			(* Löschen der Kraftwerte in den beiden IST-Einpresskurven *)
			FOR i16_ku_nr := 0  TO i_MAX_KURVEN BY 1DO
				FOR i16_mp_nr := 0  TO i_MAX_MESSPUNKTE BY 1DO
					st_ausgabe.st_kurve[i16_ku_nr].arr_kraft_ist[i16_mp_nr] := 0;
					st_ausgabe.st_kurve[i16_ku_nr].arr_weg_ist[i16_mp_nr] := 0;
				END_FOR
			END_FOR

			(* Löschen der Kraftwerte in allen Stützkurven*)
			IF st_einpressen.st_einstellungen.enu_modus = STUETZKURVE THEN
				FOR i16_ku_nr := 0  TO i_MAX_KURVEN BY 1DO
					FOR i16_mp_nr := 0  TO i_MAX_MESSPUNKTE BY 1DO
						st_ausgabe.st_kurve[i16_ku_nr].arr_kraft_stuetz[i16_mp_nr] := 0;
						st_ausgabe.st_kurve[i16_ku_nr].arr_weg_stuetz[i16_mp_nr] := 0;
					END_FOR
				END_FOR
			END_IF
		END_IF

		(* Hochzählen mit der Anzahl der bestückten Pins *)
		i16_pin_nr := ST_Virtuelle_Masterachse.i16_bestueckposzaehler;
		(* Abfrage Array-Grösse auf Überlauf *)
		IF i16_pin_nr > i_MAX_KURVEN THEN
			i16_pin_nr := 0;
		END_IF

		(* Die Messpunkte werden gradgenau aufgenommen und entsprechen deshalb den Winkelgraden der Bestückachse *)
		i16_mp_nr := ui_akt_pos_bestueckachse;

		CASE st_einpressen.st_einstellungen.enu_modus OF
			KEIN_MODUS:	(* Fehler Auswahl Einpressmodus *)
				sm_fehler_einpressmodus := TRUE;
				fb_state_entry.i16_next_step := FEHLER;

			FMAX:	(* Einpressen mit Überwachung auf Maximalkraft und Sicherheitsabfrage der Minimalkraft*)
				(*st_einpressen.st_einstellungen.lr_minkraft_einpressen := 12.0;*)
				IF  lr_kraft_n > st_ausgabe.st_ergebnisse.lr_maxkraft_einpressen THEN
					st_ausgabe.st_ergebnisse.lr_maxkraft_einpressen := lr_kraft_n;
				END_IF
				(* Fehlerfall: Voreingestellte Maximalkraft überschritten nur im Automatik Betrieb *)
				IF  gi16_betriebsart = AUTO AND lr_kraft_n > lr_help_maxkraft_einpressen THEN		(*st_einpressen.st_einstellungen.lr_maxkraft_einpressen*)
					sm_aktkraft_groesser_maxkraft_einpressen := TRUE;
					fb_state_entry.i16_next_step := FEHLER;
				END_IF

				(* Fehlerfall: Voreingestellte Minimalkraft unterschritten *)
				IF	lr_weg_grad =0 THEN
					st_ausgabe.st_ergebnisse.lr_maxkraft_einpres_proHub:=0;
				END_IF
				IF  lr_kraft_n > st_ausgabe.st_ergebnisse.lr_maxkraft_einpres_proHub THEN
					st_ausgabe.st_ergebnisse.lr_maxkraft_einpres_proHub:=lr_kraft_n;
				END_IF

				IF	gi16_betriebsart = AUTO AND
					st_einpressen.st_einstellungen.lr_minkraft_einpressen > 0 AND
					nockenschaltwerk_bestueckachse.fb.arr_spur[SP_BESTUECKSCHIEBERHUB ] AND
					st_ausgabe.st_ergebnisse.lr_maxkraft_einpres_proHub < st_einpressen.st_einstellungen.lr_minkraft_einpressen	THEN
					i16_merker:=i16_merker+1;
					(*	sm_aktkraft_kleiner_minkraft_einpressen := TRUE;
						fb_state_entry.i16_next_step := FEHLER;*)
				END_IF

				(* Aufzeichnen der Überlaufkraft nach einem Einpressfehler *)
				IF  lr_kraft_n > st_ausgabe.st_ergebnisse.lr_ueberlaufkraft THEN
					st_ausgabe.st_ergebnisse.lr_ueberlaufkraft := lr_kraft_n;
				END_IF

			FMIN_FMAX:	(* Einpressen mit Überwachung von Minimal- und Maximalkraft. Der Weg spielt hier keine Rolle! *)
				(* Aktuelle Kraft gradgenau einlesen *)
				IF st_ausgabe.st_kurve[i16_pin_nr].arr_kraft_ist[i16_mp_nr] = 0 THEN
					(* Einmalig den aktuellen Kraftwert eintragen, wenn Messpunkt im Array noch leer ist *)
					st_ausgabe.st_kurve[i16_pin_nr].arr_kraft_ist[i16_mp_nr] := lr_kraft_n;
				END_IF

				(* Aufnehmen der maximal aufgetretenen Kraft *)
				IF st_ausgabe.st_kurve[i16_pin_nr].arr_kraft_ist[i16_mp_nr] > st_ausgabe.st_ergebnisse.lr_maxkraft_einpressen THEN
					st_ausgabe.st_ergebnisse.lr_maxkraft_einpressen := st_ausgabe.st_kurve[i16_pin_nr].arr_kraft_ist[i16_mp_nr];
				END_IF

				(* Fehlerfall: Überwachen der Maximalkraft beim Aufnahmehub *)
				IF 	nockenschaltwerk_bestueckachse.fb.arr_spur[SP_AUFNAHMEHUB ] AND
					st_ausgabe.st_kurve[i16_pin_nr].arr_kraft_ist[i16_mp_nr] > 0
					THEN
						IF st_ausgabe.st_kurve[i16_pin_nr].arr_kraft_ist[i16_mp_nr] > st_einpressen.st_einstellungen.lr_maxkraft_aufnahme THEN
							st_einpressen.st_einstellungen.lr_maxkraft_aufnahme := st_ausgabe.st_kurve[i16_pin_nr].arr_kraft_ist[i16_mp_nr];
							sm_aktkraft_groesser_maxkraft_aufnahme := TRUE;
							fb_state_entry.i16_next_step := FEHLER;
						END_IF
				END_IF

				(* Fehlerfall: Überwachen der Maximalkraft beim Auftreffen des Pins auf den Isolierkörper *)
				IF 	nockenschaltwerk_bestueckachse.fb.arr_spur[SP_EINPRESSHUB ] AND
					st_ausgabe.st_kurve[i16_pin_nr].arr_kraft_ist[i16_mp_nr] > 0
					THEN
						IF st_ausgabe.st_kurve[i16_pin_nr].arr_kraft_ist[i16_mp_nr] > st_einpressen.st_einstellungen.lr_maxkraft_einpressen THEN
							st_einpressen.st_einstellungen.lr_maxkraft_einpressen := st_ausgabe.st_kurve[i16_pin_nr].arr_kraft_ist[i16_mp_nr];
							sm_aktkraft_groesser_maxkraft_einpressen := TRUE;
							fb_state_entry.i16_next_step := FEHLER;
						END_IF
				END_IF

				(* Fehlerfall: Überwachen der Minimalkraft beim Einpresshub *)
				IF 	nockenschaltwerk_bestueckachse.fb.arr_spur[SP_MIN_KRAFT_EINPRESSEN ] AND
					st_ausgabe.st_kurve[i16_pin_nr].arr_kraft_ist[i16_mp_nr] > 0
					THEN
						IF st_ausgabe.st_kurve[i16_pin_nr].arr_kraft_ist[i16_mp_nr] < st_einpressen.st_einstellungen.lr_minkraft_einpressen THEN
							st_einpressen.st_einstellungen.lr_minkraft_einpressen := st_ausgabe.st_kurve[i16_pin_nr].arr_kraft_ist[i16_mp_nr];
							sm_aktkraft_kleiner_minkraft_einpressen := TRUE;
							fb_state_entry.i16_next_step := FEHLER;
						END_IF
				END_IF

			HUELLKURVE:	(* Einpressen mit Hüllkurve um Stützkurve*)
				(* Aktuelle Kraft in die Ist-Kurve einlesen *)
				IF st_ausgabe.st_kurve[i16_pin_nr].arr_kraft_ist[i16_mp_nr] = 0 THEN
					(* Einmalig den aktuellen Kraftwert eintragen, wenn Messpunkt im Array noch leer ist *)
					st_ausgabe.st_kurve[i16_pin_nr].arr_kraft_ist[i16_mp_nr] := lr_kraft_n;
				END_IF
				(* Aktuellen Weg in die Ist-Kurve einlesen, wobei in diesem Fall das Arrayelement dem aktuellen Winkel entspricht. *)
				IF st_ausgabe.st_kurve[i16_pin_nr].arr_weg_ist[i16_mp_nr] = 0 THEN
					(* Einmalig den aktuellen Wegwert eintragen, wenn Messpunkt im Array noch leer ist *)
					st_ausgabe.st_kurve[i16_pin_nr].arr_weg_ist[i16_mp_nr] := lr_weg_grad;
				END_IF

				(* Toleranzabfrage und Fehlerauswertung *)
				IF st_ausgabe.st_kurve[i16_pin_nr].arr_kraft_ist[i16_mp_nr] > 0 AND st_ausgabe.st_kurve[i16_pin_nr].arr_weg_ist[i16_mp_nr] > 0 THEN
					b_kraft_weg_in_mp_ok := FALSE;
					(* Werte sind gültig -> Abfrage , ob Kraft und Weg im Toleranzrechteck liegen. *)
					FOR i16_mp_nr := 0  TO i_MAX_MESSPUNKTE BY 1DO
						IF	st_ausgabe.st_kurve[i16_pin_nr].arr_kraft_ist[i16_mp_nr] >= (st_ausgabe.st_kurve[i16_pin_nr].arr_kraft_ist[i16_mp_nr] - st_einpressen.st_einstellungen.lr_delta_kraft) AND
							st_ausgabe.st_kurve[i16_pin_nr].arr_kraft_ist[i16_mp_nr] <= (st_ausgabe.st_kurve[i16_pin_nr].arr_kraft_ist[i16_mp_nr] + st_einpressen.st_einstellungen.lr_delta_kraft) AND
							st_ausgabe.st_kurve[i16_pin_nr].arr_weg_ist[i16_mp_nr] >= (st_ausgabe.st_kurve[i16_pin_nr].arr_weg_ist[i16_mp_nr] - st_einpressen.st_einstellungen.lr_delta_weg) AND
							st_ausgabe.st_kurve[i16_pin_nr].arr_weg_ist[i16_mp_nr] <= (st_ausgabe.st_kurve[i16_pin_nr].arr_weg_ist[i16_mp_nr] + st_einpressen.st_einstellungen.lr_delta_weg)
							THEN
								b_kraft_weg_in_mp_ok := TRUE;
								EXIT;
						ELSE
							b_kraft_weg_in_mp_ok := FALSE;
						END_IF
					END_FOR

					(* Fehlerfall: Aktueller Messpunkt liegt mit seiner Kraft oder seinem Weg nicht im Toleranzrechteck *)
					IF NOT b_kraft_weg_in_mp_ok THEN
						sm_kraft_weg_ausserhalb_huellkurve := TRUE;
						fb_state_entry.i16_next_step := FEHLER;
					END_IF
				END_IF

			STUETZKURVE:	(* Einlernen der Stützkurve *)
				(* Aktuelle Kraft in die Stuetzkurve einlesen *)
				IF st_ausgabe.st_kurve[i16_pin_nr].arr_kraft_stuetz[i16_mp_nr] = 0 THEN
					(* Einmalig den aktuellen Kraftwert eintragen, wenn Messpunkt im Array noch leer ist *)
					st_ausgabe.st_kurve[i16_pin_nr].arr_kraft_stuetz[i16_mp_nr] := lr_kraft_n;
				END_IF
				(* Aktuellen Weg in die Stuetzkurve einlesen, wobei in diesem Fall das Arrayelement dem aktuellen Winkel entspricht. *)
				IF st_ausgabe.st_kurve[i16_pin_nr].arr_weg_stuetz[i16_mp_nr] = 0 THEN
					(* Einmalig den aktuellen Wegwert eintragen, wenn Messpunkt im Array noch leer ist *)
					st_ausgabe.st_kurve[i16_pin_nr].arr_weg_stuetz[i16_mp_nr] := lr_weg_grad;
				END_IF
		END_CASE

		(* Manuelle Messbereichsumschaltung anhand des Einstellwertes für Maximalkraft beim Einpressen. *)
		IF gst_datensatz.st_band.st_einpressen.st_einstellungen.lr_maxkraft_einpressen > (i_KRAFTFAKTOR_MB1 * 0.75) THEN
			a_messbereich_1_oder_2 := TRUE;
		ELSE
			(* Automatische Messbereichsumschaltung, wenn die maximale Einpresskraft 75% des Messbereichsendwertes überschreitet. *)
			IF st_ausgabe.st_ergebnisse.lr_maxkraft_einpressen > (i_KRAFTFAKTOR_MB1 * 0.75) THEN
				a_messbereich_1_oder_2 := TRUE;
			END_IF
		END_IF

		(*-----------------------Weiterschaltbedingungen----------------------------*)
		IF NOT st_ctrl_in.b_start THEN
			(* Messbereichsanpassung nur, wenn die Krafteinstellung für maximale Einpresskraft es erlaubt. *)
			IF gst_datensatz.st_band.st_einpressen.st_einstellungen.lr_maxkraft_einpressen < (i_KRAFTFAKTOR_MB1 * 0.75) THEN
				(* Automatische Messbereichsumschaltung, wenn die maximale Einpresskraft 50% des Messbereichsendwertes unterschreitet. *)
				IF st_ausgabe.st_ergebnisse.lr_maxkraft_einpressen < (i_KRAFTFAKTOR_MB1 * 0.5) THEN
					a_messbereich_1_oder_2 := FALSE;
				END_IF
			END_IF
			a_start_messung := FALSE;
			fb_state_entry.i16_next_step := BEREIT;
		END_IF

(*=======================================================*)
	FEHLER:
		IF fb_state_entry.E THEN
			st_ctrl_out.b_fehler := TRUE;
			fb_ton_quitt.IN := FALSE;
		END_IF

		(* Aufzeichnen der Überlaufkraft nach einem Einpressfehler *)
		IF  lr_kraft_n > st_ausgabe.st_ergebnisse.lr_ueberlaufkraft THEN
			st_ausgabe.st_ergebnisse.lr_ueberlaufkraft := lr_kraft_n;
		END_IF

		(*-----------------------Weiterschaltbedingungen----------------------------*)
		IF st_ctrl_in.b_quitt AND NOT fb_state_entry.E THEN
			st_ctrl_out.b_fehler := FALSE;
			fb_ton_quitt.IN := TRUE;
		END_IF

		IF fb_ton_quitt.Q THEN
			fb_ton_quitt.IN := FALSE;
			fb_state_entry.i16_next_step := INIT;
		END_IF

(*=======================================================*)
	STOP:
		IF fb_state_entry.E THEN
			fb_ton_quitt.IN := FALSE;
		END_IF

		(*-----------------------Weiterschaltbedingungen----------------------------*)
		IF st_ctrl_in.b_quitt AND NOT fb_state_entry.E THEN
			fb_ton_quitt.IN := TRUE;
		END_IF

		IF fb_ton_quitt.Q THEN
			fb_ton_quitt.IN := FALSE;
			fb_state_entry.i16_next_step := INIT;
		END_IF
END_CASE

fb_state_entry(
	i16_next_step:= ,
	i16_pos:= 2,
	s_debugtext:= ,
	E=> , 
	X=> ,
	i16_step=> ,
	i16_last_step=> );

(* Fehlermeldungen und Betriebsmeldungen ab dem Startindex in die globalen Meldungsarrays schreiben *)
garr_stoermeldungen[st_config.i16_meld_startindex + 0] := sm_fehler_einpressmodus;
garr_stoermeldungen[st_config.i16_meld_startindex + 1] := sm_aktkraft_groesser_maxkraft_aufnahme;
garr_stoermeldungen[st_config.i16_meld_startindex + 2] := sm_aktkraft_groesser_maxkraft_einpressen;
garr_stoermeldungen[st_config.i16_meld_startindex + 3] := sm_aktkraft_kleiner_minkraft_einpressen;
garr_stoermeldungen[st_config.i16_meld_startindex + 4] := sm_kraft_weg_ausserhalb_huellkurve;
garr_stoermeldungen[st_config.i16_meld_startindex + 5] := sm_fehler_analogwert_kraftmessdose;
garr_stoermeldungen[st_config.i16_meld_startindex + 6] := sm_max_mb_ueberschritten;
garr_stoermeldungen[st_config.i16_meld_startindex + 7] := sm_max_einstell_mb_ueberschritten;
garr_stoermeldungen[st_config.i16_meld_startindex + 8] := FALSE;
garr_stoermeldungen[st_config.i16_meld_startindex + 9] := FALSE;
garr_stoermeldungen[st_config.i16_meld_startindex + 10] := FALSE;
garr_stoermeldungen[st_config.i16_meld_startindex + 11] := FALSE;
garr_stoermeldungen[st_config.i16_meld_startindex + 12] := FALSE;
garr_stoermeldungen[st_config.i16_meld_startindex + 13] := FALSE;
garr_stoermeldungen[st_config.i16_meld_startindex + 14] := FALSE;
garr_stoermeldungen[st_config.i16_meld_startindex + 15] := FALSE;
garr_stoermeldungen[st_config.i16_meld_startindex + 16] := FALSE;
garr_stoermeldungen[st_config.i16_meld_startindex + 17] := FALSE;
garr_stoermeldungen[st_config.i16_meld_startindex + 18] := FALSE;
garr_stoermeldungen[st_config.i16_meld_startindex + 19] := FALSE;

garr_betriebsmeldungen[st_config.i16_meld_startindex + 0] := FALSE;
garr_betriebsmeldungen[st_config.i16_meld_startindex + 1] := FALSE;
garr_betriebsmeldungen[st_config.i16_meld_startindex + 2] := FALSE;
garr_betriebsmeldungen[st_config.i16_meld_startindex + 3] := FALSE;
garr_betriebsmeldungen[st_config.i16_meld_startindex + 4] := FALSE;
garr_betriebsmeldungen[st_config.i16_meld_startindex + 5] := FALSE;
garr_betriebsmeldungen[st_config.i16_meld_startindex + 6] := FALSE;
garr_betriebsmeldungen[st_config.i16_meld_startindex + 7] := FALSE;
garr_betriebsmeldungen[st_config.i16_meld_startindex + 8] := FALSE;
garr_betriebsmeldungen[st_config.i16_meld_startindex + 9] := FALSE;
garr_betriebsmeldungen[st_config.i16_meld_startindex + 10] := FALSE;
garr_betriebsmeldungen[st_config.i16_meld_startindex + 11] := FALSE;
garr_betriebsmeldungen[st_config.i16_meld_startindex + 12] := FALSE;
garr_betriebsmeldungen[st_config.i16_meld_startindex + 13] := FALSE;
garr_betriebsmeldungen[st_config.i16_meld_startindex + 14] := FALSE;
garr_betriebsmeldungen[st_config.i16_meld_startindex + 15] := FALSE;
garr_betriebsmeldungen[st_config.i16_meld_startindex + 16] := FALSE;
garr_betriebsmeldungen[st_config.i16_meld_startindex + 17] := FALSE;
garr_betriebsmeldungen[st_config.i16_meld_startindex + 18] := FALSE;
garr_betriebsmeldungen[st_config.i16_meld_startindex + 19] := FALSE;
END_PROGRAM

(* POU EPT Lib/CamEditor/Verfahrberechnungen/ST_MFCalcConstPhase, ST *)
FUNCTION_BLOCK ST_MFCalcConstPhase
VAR_INPUT
	st_config								: struct_config;
	st_ctrl_in								: struct_ctrl_in;

	(* Kurvenscheibendaten *)
	udiTableId							: MC_CAM_ID;			(* Table-ID *)
	eMotionFunctionType					: MC_MotionFunctionType;	(*Bewegungsgesetz: MOTIONFUNCTYPE_POLYNOM5 etc.*)
	i16_startpunkt_edit_mf_tab				: INT;
	arr_db_mf_tab						: ARRAY[1..i_MAX_NUM_MFP] OF struct_db_motionfunctionpoint;	(* Vorgabe aus der Datenbank *)

	(* Bewegungsdaten an der Last *)
	lrVeloMax							: LREAL;	(*maximale Geschwindigkeit [mm/s] an der Last *)
	lrAccMax								: LREAL;	(*maximale Beschleunigung [mm/s²] an der Last *)
	lrDecMax							: LREAL;	(*maximale Beschleunigung [mm/s²] an der Last *)

	lrModuloValue 						: LREAL ;
END_VAR
VAR_IN_OUT
	st_AxisRefMaster						: AXIS_REF;
	st_AxisRefSlave						: AXIS_REF;
END_VAR
VAR_OUTPUT
	lrMasterVeloMax						: LREAL;	(* Maximum Master Velocity [°/s] *)
	lrMasterRotPerMinMax					: LREAL;	(* Maximum Master Rotations per Minute [1/min] *)
	st_ctrl_out							: struct_ctrl_out;
END_VAR
VAR
	st_sm						 		: struct_cameditor_meldungen;
	fb_state_entry							: ST_StateEntry;
	fb_ton_quitt							: TON;
	fb_ton_wz							: TON;

	stMotionFunctionPointDummy			: MC_MotionFunctionPoint;	(* Dummy-Punkt *)
(*	TYPE MC_MotionFunctionPoint :
		STRUCT
		    PointIndex        		: MC_MotionFunctionPoint_ID;
		    FunctionType   		: MC_MotionFunctionType;
		    PointType         		: MC_MotionPointType;
		    RelIndexNextPoint 	: MC_MotionFunctionPoint_ID;
		    MasterPos         		: LREAL; (* X *)
		    SlavePos          		: LREAL; (* Y *)
		    SlaveVelo         		: LREAL; (* Y' *)
		    SlaveAcc          		: LREAL; (* Y'' *)
		    SlaveJerk         		: LREAL; (* Y''' *)
		END_STRUCT
	END_TYPE
*)

	(*Motion Function runterschreiben an NC*)
	astWriteMotionFunction 				: ARRAY[1..i_MAX_NUM_MFP] OF MC_MotionFunctionPoint;
	stWriteMFCamTableRef				: MC_CAM_Ref;	(*Definition Zieltabelle*)
	fbCamTableSelect					: MC_CamTableSelect;
	fbWriteMF							: MC_WriteMotionFunction;
	b_cam_table_select_periodic			: BOOL := FALSE;
	b_cam_table_select_master_absolute	: BOOL := FALSE;
	b_cam_table_select_slave_absolute		: BOOL := FALSE;

	(*Motion Function hochladen von NC*)
	fbReadMF							: MC_ReadMotionFunction;
	stReadMFCamTableRef				: MC_CAM_Ref;	(*Definition Zieltabelle*)
	astReadMotionFunction 				: ARRAY[0..i_MAX_NUM_MFP] OF MC_MotionFunctionPoint;

	(*Berechnung Konstantfahrphase*)
	fbMFcalcConstVelo					: ST_MFcalcConstVelo;	(*Baustein zur Berechnung, ob eine Konstantfahphase möglich ist*)
	stDataCalcConstVelo 					: ARRAY[1..4] OF MC_MotionFunctionPoint;	(*Aus der Berechnung ermittelte Punktedaten*)

	(* Berechnung Mastergeschwindigkeit*)
	fbMFMaxMasterVelo					: ST_MFMaxMasterVelo;	(* Baustein zur Berechnung der maximalen Mastergeschwindigkeit *)

	(*Temporäre Variablen *)
	iPointCount							: INT := 0;
	iNumMfPoints							: INT := 0;
	i_point_nr							: INT := 0;
	err_id								: UDINT := 0;
	i16_anzahl_mfps						: INT;
	lrStartPointMaster						: LREAL;	(* Startpunkt Master [°] *)
	lrStartPointSlave						: LREAL;	(* Startpunkt Slave [mm] *)
	lrEndPointMaster						: LREAL;	(* Endpunkt Master [°] *)
	lrEndPointSlave						: LREAL;	(* Endpunkt Slave [mm] *)
	lr_anfang_cam_table					: LREAL := 0;	(* Anfang Darstellungsbereich MF-Tabelle *)
	lr_ende_cam_table					: LREAL := 0;	(* Ende Darstellungsbereich MF-Tabelle *)
END_VAR
VAR CONSTANT
	i_MAX_NUM_MFP						: INT := 100;
END_VAR
fb_ton_wz(IN:= , PT:= , Q=> , ET=> );
fb_ton_quitt(IN:= , PT:= t#50ms, Q=> , ET=> );

(* ======================================Schrittkette======================================== *)
fb_state_entry(
	i16_next_step:= ,
	i16_pos:= 1,
	s_debugtext:= ,
	E=> ,
	X=> ,
	i16_step=> ,
	i16_last_step=> );

CASE fb_state_entry.i16_step OF
(*=======================================================*)
	0:	(* Init *)
		st_ctrl_out.b_bereit := FALSE;
		st_ctrl_out.b_fertig := FALSE;
		st_ctrl_out.b_fehler := FALSE;
		fbCamTableSelect.Execute := FALSE;
		fbWriteMF.Execute := FALSE;
		fbReadMF.Execute := FALSE;
		fbMFMaxMasterVelo.bExecute := FALSE;
		fbMFcalcConstVelo.bExecute := FALSE;
		err_id := 0;
		i16_anzahl_mfps := 0;
		st_sm.berechne_konstantfahrphase := FALSE;
		st_sm.berechne_max_master_geschwindigkeit := FALSE;
		st_sm.lese_camtable := FALSE;
		st_sm.lese_mfp := FALSE;
		st_sm.lesen_werte_mf_tab := FALSE;
		st_sm.schreibe_camtable := FALSE;
		st_sm.schreibe_mfp := FALSE;

		fb_state_entry.i16_next_step := 10;

(*=======================================================*)
	10:	(* Warte auf Start *)
		IF lrModuloValue > 0 THEN
			b_cam_table_select_periodic := TRUE;
			b_cam_table_select_master_absolute := TRUE;
			b_cam_table_select_slave_absolute := FALSE;
		ELSE
			b_cam_table_select_periodic := FALSE;
			b_cam_table_select_master_absolute := TRUE;
			b_cam_table_select_slave_absolute := TRUE;
		END_IF

		(*-----------------------Weiterschaltbedingungen----------------------------*)
		IF st_ctrl_in.b_start THEN
			i16_anzahl_mfps := 0;
			lrMasterVeloMax := 0;
			lrMasterRotPerMinMax := 0;
			fb_state_entry.i16_next_step := 100;
		END_IF

(*=======================================================*)
	100:	(*  *)
		IF fb_state_entry.E THEN
			FOR i_point_nr := 1 TO i_MAX_NUM_MFP BY 1 DO
				(*Für Download: Initialisieren aller  MFPs im Array *)
				astWriteMotionFunction[i_point_nr] := stMotionFunctionPointDummy;
				astWriteMotionFunction[i_point_nr].RelIndexNextPoint  := 1;

				(* Übernahme der Daten aus der WKZ-Datenbank *)
				astWriteMotionFunction[i_point_nr].FunctionType := arr_db_mf_tab[i_point_nr].FunctionType;
				astWriteMotionFunction[i_point_nr].MasterPos  := arr_db_mf_tab[i_point_nr].MasterPos;
				astWriteMotionFunction[i_point_nr].SlavePos  := arr_db_mf_tab[i_point_nr].SlavePos;
				astWriteMotionFunction[i_point_nr].PointType  := arr_db_mf_tab[i_point_nr].PointType;
				astWriteMotionFunction[i_point_nr].PointIndex  := arr_db_mf_tab[i_point_nr].PointIndex;

				IF astWriteMotionFunction[i_point_nr].FunctionType > MOTIONFUNCTYPE_NOTDEF THEN
					i16_anzahl_mfps := i16_anzahl_mfps + 1;
				END_IF
			END_FOR

			(* Beim Letzen Punkt in der Tabelle immer den RelIndexNextPoint auf 0 setzen *)
			astWriteMotionFunction[i16_anzahl_mfps].RelIndexNextPoint := 0;

			(* Darstellungsbereich der MF-Tabelle (wird benötigt für die Funktion "MC_ReadMotionFunctionValues") *)
			IF lrModuloValue > 0 THEN
				lr_anfang_cam_table := 0;
				lr_ende_cam_table := lrModuloValue;
			ELSE
				lr_anfang_cam_table := arr_db_mf_tab[1].MasterPos;
				lr_ende_cam_table := arr_db_mf_tab[i16_anzahl_mfps].MasterPos;
			END_IF
		END_IF

		(*-----------------------Weiterschaltbedingungen----------------------------*)
		fb_state_entry.i16_next_step := 110;


(*=======================================================*)
	110:	(* Starte Berechnung der Konstantfahrphase *)
		IF fb_state_entry.E THEN
			fbMFcalcConstVelo.bExecute := TRUE;
		END_IF

		(*-----------------------Weiterschaltbedingungen----------------------------*)
		IF fbMFcalcConstVelo.bBusy THEN
			fb_state_entry.i16_next_step := 120;
		END_IF

(*=======================================================*)
	120:	(* Starte Berechnung der Konstantfahrphase *)
		IF NOT fbMFcalcConstVelo.bBusy THEN
			IF fbMFcalcConstVelo.bDone THEN
				fbMFcalcConstVelo.bExecute := FALSE;
				IF fbMFcalcConstVelo.bConstantVelo THEN
					iNumMfPoints := i16_anzahl_mfps + 2;
					fb_state_entry.i16_next_step := 130;
				ELSE
					iNumMfPoints := i16_anzahl_mfps;
					fb_state_entry.i16_next_step := 140;
				END_IF
			ELSIF fbMFcalcConstVelo.bError THEN
				st_sm.berechne_konstantfahrphase := TRUE;
				fb_state_entry.i16_next_step := 1000;
			END_IF
		END_IF

(*=======================================================*)
	130:	(* Auswertung ob Konstantfahrphase *)
		IF fb_state_entry.E THEN
			(* Verschieben aller weiteren Punkte um 2 Positionen nach hinten *)
			FOR i_point_nr := iNumMfPoints TO (i16_startpunkt_edit_mf_tab + 1) BY -1 DO
				astWriteMotionFunction[i_point_nr] := astWriteMotionFunction[i_point_nr - 2];
				astWriteMotionFunction[i_point_nr].PointIndex := i_point_nr;
			END_FOR

			iPointCount := i16_startpunkt_edit_mf_tab;

			(*Startpunkt: spezifische Daten anpassen*)
			astWriteMotionFunction[iPointCount].MasterPos := stDataCalcConstVelo[1].MasterPos;
			astWriteMotionFunction[iPointCount].SlavePos := stDataCalcConstVelo[1].SlavePos;
			astWriteMotionFunction[iPointCount].SlaveVelo := stDataCalcConstVelo[1].SlaveVelo;
			astWriteMotionFunction[iPointCount].SlaveJerk := stDataCalcConstVelo[1].SlaveJerk;
			(*Punktetyp eintragen*)
			astWriteMotionFunction[iPointCount].RelIndexNextPoint := 1;
			astWriteMotionFunction[iPointCount].FunctionType := stDataCalcConstVelo[1].FunctionType;
			astWriteMotionFunction[iPointCount].PointIndex := iPointCount;
			astWriteMotionFunction[iPointCount].PointType := stDataCalcConstVelo[1].PointType;

			iPointCount := iPointCount + 1;

			(*Zwischenpunkt 1: Konstantfahrphase eintragen*)
			astWriteMotionFunction[iPointCount].MasterPos := stDataCalcConstVelo[2].MasterPos;
			astWriteMotionFunction[iPointCount].SlavePos := stDataCalcConstVelo[2].SlavePos;
			astWriteMotionFunction[iPointCount].SlaveVelo := stDataCalcConstVelo[2].SlaveVelo;
			astWriteMotionFunction[iPointCount].SlaveJerk := stDataCalcConstVelo[2].SlaveJerk;
			(*Punktetyp eintragen*)
			astWriteMotionFunction[iPointCount].RelIndexNextPoint := 1;
			astWriteMotionFunction[iPointCount].FunctionType := stDataCalcConstVelo[2].FunctionType;
			astWriteMotionFunction[iPointCount].PointIndex := iPointCount;
			astWriteMotionFunction[iPointCount].PointType := stDataCalcConstVelo[2].PointType;
	
			iPointCount := iPointCount + 1;
	
			(*Zwischenpunkt 2: Konstantfahrphase eintragen*)
			astWriteMotionFunction[iPointCount].MasterPos := stDataCalcConstVelo[3].MasterPos;
			astWriteMotionFunction[iPointCount].SlavePos := stDataCalcConstVelo[3].SlavePos;
			astWriteMotionFunction[iPointCount].SlaveVelo := stDataCalcConstVelo[3].SlaveVelo;
			astWriteMotionFunction[iPointCount].SlaveJerk := stDataCalcConstVelo[3].SlaveJerk;
			(*Punktetyp eintragen*)
			astWriteMotionFunction[iPointCount].RelIndexNextPoint := 1;
			astWriteMotionFunction[iPointCount].FunctionType := stDataCalcConstVelo[3].FunctionType;
			astWriteMotionFunction[iPointCount].PointIndex := iPointCount;
			astWriteMotionFunction[iPointCount].PointType := stDataCalcConstVelo[3].PointType;

			iPointCount := iPointCount + 1;

			(* Beim Letzen Punkt in der Tabelle immer den RelIndexNextPoint auf 0 setzen *)
			astWriteMotionFunction[i16_anzahl_mfps + 2].RelIndexNextPoint := 0;
		END_IF

		(*-----------------------Weiterschaltbedingungen----------------------------*)
		fb_state_entry.i16_next_step := 140;

(*=======================================================*)
	140:	(* Alle Punkte der MF-Tabelle werden an die NC runter geschrieben  *)
		IF fb_state_entry.E THEN
			(*Tabelle initialisieren *)
			stWriteMFCamTableRef.pArray := ADR(astWriteMotionFunction[1]);	(* Adresse des ersten eindimensionalen Arrays vom Typ MC_MotionFunctionPoint. Jedes Array-Element enthält eine Beschreibung einer Stützstelle der Kurvenscheibe. *)
			stWriteMFCamTableRef.ArraySize := SIZEOF(astWriteMotionFunction[1]) * iNumMfPoints;
			stWriteMFCamTableRef.TableType := MC_TABLETYPE_MOTIONFUNCTION;
			stWriteMFCamTableRef.NoOfColumns := 1;	(* Bei Table Type "MC_TABLETYPE_MOTIONFUNCTION" ist NoOfColumns immer 1 *)
			stWriteMFCamTableRef.NoOfRows := iNumMfPoints;

			fbCamTableSelect.Execute := TRUE;
		END_IF

		(*-----------------------Weiterschaltbedingungen----------------------------*)
		IF fbCamTableSelect.Busy THEN
			fb_state_entry.i16_next_step := 150;
		END_IF

(*=======================================================*)
	150:	(* Alle Punkte der MF-Tabelle werden an die NC runter geschrieben  *)
		IF NOT fbCamTableSelect.Busy THEN
			IF fbCamTableSelect.Done THEN
				fbCamTableSelect.Execute := FALSE;
				fb_state_entry.i16_next_step := 200;
			ELSIF fbCamTableSelect.Error THEN
				st_sm.schreibe_camtable := TRUE;
				err_id := fbCamTableSelect.ErrorID;
				fb_state_entry.i16_next_step := 1000;
			END_IF
		END_IF

(*=======================================================*)
	200:	(* Lesen der MF-Tabelle von der NC  *)
		IF fb_state_entry.E THEN
			stReadMFCamTableRef.pArray := ADR(astReadMotionFunction[0]);
			stReadMFCamTableRef.ArraySize := SIZEOF(astReadMotionFunction[0]) * (iNumMfPoints + 1) ;
			stReadMFCamTableRef.NoOfColumns := 2;		(* Master und Slave Spalte*)
			stReadMFCamTableRef.NoOfRows := iNumMfPoints;
			stReadMFCamTableRef.TableType := MC_TABLETYPE_MOTIONFUNCTION;
			
			(* Für Upload initialisieren *)
			FOR iPointCount := 1 TO i_MAX_NUM_MFP DO
				astReadMotionFunction[iPointCount] := stMotionFunctionPointDummy;
			END_FOR

			fbReadMF.Execute := TRUE;
		END_IF

		(*-----------------------Weiterschaltbedingungen----------------------------*)
		IF fbReadMF.Busy THEN
			fb_state_entry.i16_next_step := 210;
		END_IF

(*=======================================================*)
	210:	(* Die gesamte MF-Tabelle hochladen  *)
		IF NOT fbReadMF.Busy THEN
			IF fbReadMF.Done THEN
				fbReadMF.Execute := FALSE;
				fb_state_entry.i16_next_step := 220;
			ELSIF fbReadMF.Error THEN
				st_sm.lese_camtable := TRUE;
				err_id := fbReadMF.ErrorID;
				fb_state_entry.i16_next_step := 1000;
			END_IF
		END_IF

(*=======================================================*)
	220:	(* Grenzhubzahlberechung  *)
		IF fb_state_entry.E THEN
			fbMFMaxMasterVelo.bExecute := TRUE;
		END_IF

		(*-----------------------Weiterschaltbedingungen----------------------------*)
		IF fbMFMaxMasterVelo.bBusy THEN
			fb_state_entry.i16_next_step := 230;
		END_IF

(*=======================================================*)
	230:	(* Berechnung fertig  *)
		IF NOT fbMFMaxMasterVelo.bBusy THEN
			IF fbMFMaxMasterVelo.bDone THEN
				fbMFMaxMasterVelo.bExecute := FALSE;
				fb_state_entry.i16_next_step := 240;
			ELSIF fbMFMaxMasterVelo.bError THEN
				st_sm.berechne_max_master_geschwindigkeit := TRUE;
				err_id := fbMFMaxMasterVelo.udiErrorId;
				fb_state_entry.i16_next_step := 1000;
			END_IF
		END_IF

(*=======================================================*)
	240:	(* Zuweisung der maximalen Mastergeschwindigkeit *)
		IF fb_state_entry.E THEN
			lrMasterVeloMax := fbMFMaxMasterVelo.lrMasterVeloMax;
			IF lrModuloValue > 0 THEN
				lrMasterRotPerMinMax := 60.0 * lrMasterVeloMax / lrModuloValue;
			ELSE
				lrMasterRotPerMinMax := 0;
			END_IF
		END_IF

		(*-----------------------Weiterschaltbedingungen----------------------------*)
		fb_state_entry.i16_next_step := 250;

(*=======================================================*)
	250:	(* Fertig  *)
		IF fb_state_entry.E THEN
			st_ctrl_out.b_fertig := TRUE;
		END_IF

		(*-----------------------Weiterschaltbedingungen----------------------------*)
		IF NOT st_ctrl_in.b_start THEN
			st_ctrl_out.b_fertig := FALSE;
			fb_state_entry.i16_next_step := 10;
		END_IF

(*=======================================================*)
	FEHLER: (* Fehler *)
		IF fb_state_entry.E THEN
			st_ctrl_out.b_fehler := TRUE;
			fb_ton_quitt.IN := FALSE;
		END_IF

		(*-----------------------Weiterschaltbedingungen----------------------------*)
		IF st_ctrl_in.b_quitt AND NOT fb_state_entry.E THEN
			st_ctrl_out.b_fehler := FALSE;
			fb_ton_quitt.IN := TRUE;
		END_IF

		IF fb_ton_quitt.Q THEN
			fb_ton_quitt.IN := FALSE;
			fb_state_entry.i16_next_step := 0;
		END_IF
END_CASE

fb_state_entry(
	i16_next_step:= ,
	i16_pos:= 2,
	s_debugtext:= ,
	E=> ,
	X=> ,
	i16_step=> ,
	i16_last_step=> );

(* Erstellen einer neuen MF-Tabelle mit anschliessendem Füllen der Punktdaten: *)
(* Es wird eine neue Tabelle in der NC angelegt zudem werden  Master und Slave Achsen zugeordnet. *)
(* Die Länge der Tabelle mit ihren Punktdaten wird gleichzeitig mit reingeschrieben. *)
fbCamTableSelect(
	Execute:= , 
	Periodic:= b_cam_table_select_periodic,
	MasterAbsolute:= b_cam_table_select_master_absolute,
	SlaveAbsolute:= b_cam_table_select_slave_absolute,
	CamTableID:= udiTableId,
	Master := st_AxisRefMaster,
	Slave := st_AxisRefSlave,
	CamTable:= stWriteMFCamTableRef,
	Done=> ,
	Busy=> , 
	Error=> , 
	ErrorID=> );

(* Die gesamte Tabelle einlesen aus der NC *)
fbReadMF(
	Execute:= ,
	CamTableID:= udiTableId,
	PointID:= 1,
	NumPoints:= stReadMFCamTableRef.NoOfRows,
	CamTable:= stReadMFCamTableRef,
	Done=> ,
	Busy=> ,
	Error=> ,
	ErrorID=> ,
	NumPointsRead=> );

(* Die ganze oder einen Teil der MF-Tabelle schreiben *)
fbWriteMF(
	Execute:= ,
	CamTableID:= udiTableId,
	PointID:= i16_startpunkt_edit_mf_tab,
	NumPoints:= i16_anzahl_mfps,
	CamTable:= stWriteMFCamTableRef,
	Done=> ,
	Busy=> , 
	Error=> , 
	ErrorID=> );

(* Berechnen ob Konstantfahrphase möglich *)
fbMFcalcConstVelo(
	bExecute:= ,
	eMotionFunctionType:= eMotionFunctionType,
	lrStartPointMaster:= arr_db_mf_tab[i16_startpunkt_edit_mf_tab].MasterPos,
	lrStartPointSlave:= arr_db_mf_tab[i16_startpunkt_edit_mf_tab].SlavePos,
	lrEndPointMaster:= arr_db_mf_tab[i16_startpunkt_edit_mf_tab + 1].MasterPos,
	lrEndPointSlave:= arr_db_mf_tab[i16_startpunkt_edit_mf_tab + 1].SlavePos,
	lrVeloLimit:= lrVeloMax,
	lrAccLimit:= lrAccMax,
	lrDecLimit:= lrDecMax,
	lrModuloValue:= lrModuloValue,
	stData:= stDataCalcConstVelo,
	bDone=> ,
	bError=> ,
	szErrText=> ,
	bConstantVelo=> ,
	lrVeloRef=> ,	(* Momentan nicht verwendet *)
	lrAccRef=> );	(* Momentan nicht verwendet *)

(* Berechne maximal mögliche Mastergeschwindigkeit *)
fbMFMaxMasterVelo(
	bExecute:= ,
	bEvCamTableChar:= eMotionFunctionType = MOTIONFUNCTYPE_POLYNOM7_MM,
	udiSlaveTableId:= udiTableId,
	lrVeloMax:= lrVeloMax,
	lrAccMax:= lrAccMax,
	lrDecMax:= lrDecMax,
	i16_anzahl_mfps:= iNumMfPoints,
	lr_anfang_cam_table:= lr_anfang_cam_table,
	lr_ende_cam_table:= lr_ende_cam_table,
	bDone=> ,
	bError=> , 
	udiErrorId=> ,
	szErrText=> ,
	lrMasterVeloMax=> );

IF st_config.b_config_fertig THEN
	garr_stoermeldungen[st_config.i16_meld_startindex + 0] := st_sm.lese_mfp;
	garr_stoermeldungen[st_config.i16_meld_startindex + 1] := st_sm.lese_camtable;
	garr_stoermeldungen[st_config.i16_meld_startindex + 2] := st_sm.lesen_werte_mf_tab;
	garr_stoermeldungen[st_config.i16_meld_startindex + 3] := st_sm.schreibe_mfp;
	garr_stoermeldungen[st_config.i16_meld_startindex + 4] := st_sm.schreibe_camtable;
	garr_stoermeldungen[st_config.i16_meld_startindex + 5] := st_sm.berechne_konstantfahrphase;
	garr_stoermeldungen[st_config.i16_meld_startindex + 6] := st_sm.berechne_max_master_geschwindigkeit;
	garr_stoermeldungen[st_config.i16_meld_startindex + 7] := FALSE;
	garr_stoermeldungen[st_config.i16_meld_startindex + 8] := FALSE;
	garr_stoermeldungen[st_config.i16_meld_startindex + 9] := FALSE;
	garr_stoermeldungen[st_config.i16_meld_startindex + 10] := FALSE;
	garr_stoermeldungen[st_config.i16_meld_startindex + 11] := FALSE;
	garr_stoermeldungen[st_config.i16_meld_startindex + 12] := FALSE;
	garr_stoermeldungen[st_config.i16_meld_startindex + 13] := FALSE;
	garr_stoermeldungen[st_config.i16_meld_startindex + 14] := FALSE;
	garr_stoermeldungen[st_config.i16_meld_startindex + 15] := FALSE;
	garr_stoermeldungen[st_config.i16_meld_startindex + 16] := FALSE;
	garr_stoermeldungen[st_config.i16_meld_startindex + 17] := FALSE;
	garr_stoermeldungen[st_config.i16_meld_startindex + 18] := FALSE;
	garr_stoermeldungen[st_config.i16_meld_startindex + 19] := FALSE;
	
	garr_betriebsmeldungen[st_config.i16_meld_startindex + 0] := FALSE;
	garr_betriebsmeldungen[st_config.i16_meld_startindex + 1] := FALSE;
	garr_betriebsmeldungen[st_config.i16_meld_startindex + 2] := FALSE;
	garr_betriebsmeldungen[st_config.i16_meld_startindex + 3] := FALSE;
	garr_betriebsmeldungen[st_config.i16_meld_startindex + 4] := FALSE;
	garr_betriebsmeldungen[st_config.i16_meld_startindex + 5] := FALSE;
	garr_betriebsmeldungen[st_config.i16_meld_startindex + 6] := FALSE;
	garr_betriebsmeldungen[st_config.i16_meld_startindex + 7] := FALSE;
	garr_betriebsmeldungen[st_config.i16_meld_startindex + 8] := FALSE;
	garr_betriebsmeldungen[st_config.i16_meld_startindex + 9] := FALSE;
	garr_betriebsmeldungen[st_config.i16_meld_startindex + 10] := FALSE;
	garr_betriebsmeldungen[st_config.i16_meld_startindex + 11] := FALSE;
	garr_betriebsmeldungen[st_config.i16_meld_startindex + 12] := FALSE;
	garr_betriebsmeldungen[st_config.i16_meld_startindex + 13] := FALSE;
	garr_betriebsmeldungen[st_config.i16_meld_startindex + 14] := FALSE;
	garr_betriebsmeldungen[st_config.i16_meld_startindex + 15] := FALSE;
	garr_betriebsmeldungen[st_config.i16_meld_startindex + 16] := FALSE;
	garr_betriebsmeldungen[st_config.i16_meld_startindex + 17] := FALSE;
	garr_betriebsmeldungen[st_config.i16_meld_startindex + 18] := FALSE;
	garr_betriebsmeldungen[st_config.i16_meld_startindex + 19] := FALSE;
END_IF
END_FUNCTION_BLOCK

(* POU EPT Lib/CamEditor/Verfahrberechnungen/ST_MFcalcConstVelo, ST *)
FUNCTION_BLOCK ST_MFcalcConstVelo
VAR_INPUT
	bExecute			: BOOL;
	eMotionFunctionType	: MC_MotionFunctionType;(*Bewegungsgesetz*)
	lrStartPointMaster		: LREAL;	(* Start Point Master [°] oder [mm] *)
	lrStartPointSlave		: LREAL;	(* Start Point Slave [mm] *)
	lrEndPointMaster		: LREAL;	(* End Point Master [°] oder [mm] *)
	lrEndPointSlave		: LREAL;	(* End Point Slave [mm] *)
	lrVeloLimit			: LREAL;	(*Slave Geschwindigkeitsgrenzwert [EINH/s]*)
	lrAccLimit			: LREAL;	(*Slave Beschleunigungsgrenzwert [EINH/s²]*)
	lrDecLimit			: LREAL;	(*Slave Bremsbeschleunigungsgrenzwert [EINH/s²]*)
	lrModuloValue		: LREAL;	(*Modulo-Periode des Master-Zyklus*)
END_VAR
VAR_OUTPUT
	bBusy				: BOOL;
	bDone 				: BOOL;
	bError 				: BOOL;

	bConstantVelo		: BOOL;	(* Ergebnis aus der Berechnung der Konstantfahrphase *)

	lrVeloRef			: LREAL;	(* referenced velocity *)
	lrAccRef				: LREAL;	(* referenced acceleration *)
END_VAR
VAR_IN_OUT
	stData 				: ARRAY[1..4] OF MC_MotionFunctionPoint; (*Berechnete Punktedaten*)
END_VAR
VAR
	szErrText			: STRING;		(*Error text*)
	lrVMax				: LREAL;			(*Slave Geschwindigkeit [m/s]*)
	lrAMax				: LREAL;			(*Slave Beschleunigung [m/s²]*)
	lrDMax				: LREAL;			(*Slave Verzögerung [m/s²] *)
	lrCvOrig				: LREAL;			(*Original Bewegungsgesetz*)
	lrCaOrig				: LREAL;			(*Original Bewegungsgesetz*)
	lrCv					: LREAL;			(*Polynom 5*)
	lrCa					: LREAL;			(*Polynom 5*)
	eMfType				: MC_MotionFunctionType;	(*Polynom 5*)
	lrPhiAcc				: LREAL;			(*Beschleunigungsphase*)
	lrPhiVelo				: LREAL;			(*Bewegungsphase v=const.*)
	lrPhi					: LREAL;			(*Gesamtbewegungsphase*)
	lrTAcc				: LREAL;			(*Beschleunigungszeit*)
	lrTVelo_to_TAcc		: LREAL;			(*Quotient Konstantfahrt / Beschleunigungsfahrt*)
	lrXAccOrig			: LREAL;			(*Original Beschleunigungsweg*)
	lrXAcc				: LREAL;			(*Beschleunigungsweg*)

	lrTDec				: LREAL;			(*Bremsszeit*)
	lrXDecOrig			: LREAL;			(*Original Bremssweg*)
	lrXDec				: LREAL;			(*Bremssweg*)

	lrXVelo				: LREAL;			(*Konstantfahrweg*)
	lrX					: LREAL;			(*Gesamtweg / Hub*)
	lrV					: LREAL;			(*Geschwindigkeit*)

	fb_state_entry			: ST_StateEntry;
END_VAR
(* ======================================Schrittkette======================================== *)
fb_state_entry(
	i16_next_step:= ,
	i16_pos:= 1,
	s_debugtext:= ,
	E=> ,
	X=> ,
	i16_step=> ,
	i16_last_step=> );

CASE fb_state_entry.i16_step OF
(*=======================================================*)
	0 :	(* Init*)
		bBusy := FALSE;
		bDone := FALSE;
		bError := FALSE;
		bConstantVelo := FALSE;
		szErrText := '';
		fb_state_entry.i16_next_step := 10;

(*=======================================================*)
	10:	(* Warte Execute *)

		(*-----------------------Weiterschaltbedingungen----------------------------*)
		IF bExecute THEN
			bBusy := TRUE;
			fb_state_entry.i16_next_step := 20;
		END_IF

(*=======================================================*)
	20:
		IF fb_state_entry.E THEN
			(* Die Variable lrPhi wird für lineare und runde(modulo) Master verwendet *)
 			IF lrModuloValue = 0 THEN
				(*Linearachse: Einheiten umrechnen*)
				lrX := lrEndPointSlave - lrStartPointSlave;
				lrPhi := ABS(lrEndPointMaster - lrStartPointMaster);
			ELSE
				(*Rundachse: Einheiten umrechnen*)
				lrX := lrEndPointSlave - lrStartPointSlave;
				lrPhi := MODABS(lrEndPointMaster - lrStartPointMaster, lrModuloValue);
				(* Sonderfall: phi4 - phi1 = modulowert *)
				IF (lrEndPointMaster - lrStartPointMaster = lrModuloValue) THEN
					lrPhi := lrModuloValue;
				END_IF
			END_IF

			lrVMax := lrVeloLimit;
			lrAMax := lrAccLimit;
			lrDMax := lrDecLimit;
			
			(*Bewegungsgesetz auswaehlen -> Charakteristische Werte Cv, Ca*)
			IF eMotionFunctionType = MOTIONFUNCTYPE_POLYNOM7_MM THEN
			(*Polynom 7*)
				lrCvOrig :=1.9;
				lrCaOrig :=7.51;
				eMfType := MOTIONFUNCTYPE_POLYNOM7_MM;
				lrCv :=1.9;
				lrCa :=7.51;
			
			ELSE
			(*Polynom 5*)
				lrCvOrig :=1.88;
				lrCaOrig :=5.78;
				eMfType := MOTIONFUNCTYPE_POLYNOM5_MM;
				lrCv :=1.88;
				lrCa :=5.78;
			END_IF

			(*Plausibilitaetsprüfung*)
			IF lrAMax <= 0 THEN
				fb_state_entry.i16_next_step := FEHLER;
				szErrText := 'Amax <= 0';
			ELSIF lrDMax <= 0 THEN
				fb_state_entry.i16_next_step := FEHLER;
				szErrText := 'Dmax <= 0';
			ELSIF lrVMax <= 0 THEN
				fb_state_entry.i16_next_step := FEHLER;
				szErrText := 'Vmax <= 0';
			ELSIF lrCv <= 0 THEN
				fb_state_entry.i16_next_step := FEHLER;
				szErrText := 'Cv <= 0';
			ELSIF lrCa <= 0 THEN
				fb_state_entry.i16_next_step := FEHLER;
				szErrText := 'Ca <= 0';
			ELSIF lrX = 0 THEN
				fb_state_entry.i16_next_step := FEHLER;
				szErrText := 'x = 0';
			ELSIF lrPhi <= 0 THEN
				fb_state_entry.i16_next_step := FEHLER;
				szErrText := 'phi <= 0';
			ELSE
				fb_state_entry.i16_next_step := 30;
			END_IF
		END_IF

(*=======================================================*)
	30:
		IF fb_state_entry.E THEN
			(*Berechnung: Weg, ab dem sich das Einfuegen einer Konstantfahrphase lohnt*)
			(*
			Bewegungsgesetzt der Translation: s = 0.5 * v * t = 0.5 * v^2 / a
			----------------------------------
			xAcc = 0.5 * (vmax² * Ca) / (Cv² * amax)
			xDec = 0.5 * (vmax² * Ca) / (Cv² * dmax)
			----------------------------------
			
			x		:	Gesamtweg (Hub)
			xAcc	:	Weg beim Fahren mit max. Beschleunigung, so dass die max. Geschwind. gerade erreicht wird
			xDec	:	Weg beim Fahren mit max. Verzögerung, so dass die max. Geschwind. gerade erreicht wird
			vmax	:	max. zulaessige Geschwindigkeit
			amax	:	max. zulaessige Beschleunigung
			dmax	:	max. zulaessige Verzoegerung
			Cv		:	Geschwindigkeitskennwert des Bewegungsgesetzes
			Ca		:	Beschleunigungskennwert des Bewegungsgesetzes
			*)
			
			lrXAcc := 0.5 * (lrVMax * lrVMax * lrCa) / (lrCv * lrCv * lrAMax);
			lrXAcc := F_rSign(lrX) * lrXAcc;
			lrXAccOrig := 0.5 * (lrVMax * lrVMax * lrCaOrig) / (lrCvOrig * lrCvOrig * lrAMax);
			
			lrXDec := 0.5 * (lrVMax * lrVMax * lrCa) / (lrCv * lrCv * lrDMax);
			lrXDec := F_rSign(lrX) * lrXDec;
			lrXDecOrig := 0.5 * (lrVMax * lrVMax * lrCaOrig) / (lrCvOrig * lrCvOrig * lrDMax);
			
			IF (lrXAccOrig + lrXDecOrig) < ABS(lrX) THEN
				bConstantVelo := TRUE;

				(*Berechnung Wertebereich fuer Beschleunigungsphase ohne Konstantfahrtanteil*)
				(*
				t = v / a
				--------------------------------
				tAcc = (vmax * Ca) / (Cv * amax)
				--------------------------------
				*)
				lrTAcc := (lrVMax * lrCa) / (lrAMax * lrCv);
				lrTDec := (lrVMax * lrCa) / (lrDMax * lrCv);
				(*
				---------------------------------------
				tVelo/tAcc = (x - xAcc) / (vmax * tAcc)
				---------------------------------------
				*)
				lrTVelo_to_TAcc := ABS(lrX - lrXAcc - lrXDec) / (lrVMax * (lrTAcc + lrTDec)/2);
				(*
				---------------------------------------
				tAcc = phi / {[(x - xAcc)/(vmax * tAcc)] + 1}
				---------------------------------------
				*)
				lrPhiAcc := lrPhi / (lrTVelo_to_TAcc + 1);
				lrPhiVelo := lrPhi - lrPhiAcc;

				lrXVelo := lrX - lrXAcc - lrXDec;
				lrV := lrXVelo / lrPhiVelo;

				(*Berechnete MFP Daten*)
				stData[1].FunctionType := eMfType;
				stData[1].PointType := MOTIONPOINTTYPE_VELOCITY;
				stData[1].MasterPos := lrStartPointMaster;
				stData[1].SlavePos := lrStartPointSlave;
				stData[1].SlaveVelo := lrV;
				
				stData[2].FunctionType := MOTIONFUNCTYPE_POLYNOM1;
				stData[2].PointType := MOTIONPOINTTYPE_VELOCITY;
				stData[2].MasterPos := lrStartPointMaster + (lrPhiAcc *  lrDecLimit / (lrAccLimit + lrDecLimit));
				stData[2].SlavePos := lrStartPointSlave + lrXAcc;
				stData[2].SlaveVelo := lrV;
				
				stData[3].FunctionType := eMfType;
				stData[3].PointType := MOTIONPOINTTYPE_VELOCITY;
				stData[3].MasterPos := lrEndPointMaster - (lrPhiAcc * lrAccLimit  / (lrAccLimit + lrDecLimit));
				stData[3].SlavePos := lrEndPointSlave - lrXDec;
				stData[3].SlaveVelo := lrV;
				
				stData[4].FunctionType := eMfType;
				stData[4].PointType := MOTIONPOINTTYPE_REST;
				stData[4].MasterPos := lrEndPointMaster;
				stData[4].SlavePos := lrEndPointSlave;
				stData[4].SlaveVelo := 0;
				
				lrVeloRef := ABS(lrV);
				lrAccRef := MAX(lrAccLimit,lrDecLimit) * (EXPT(lrVeloRef /lrVeloLimit,2));

			ELSE
				bConstantVelo := FALSE;
			END_IF
			fb_state_entry.i16_next_step := 40;
		END_IF

(*=======================================================*)
	40: (* Fertig *)
		IF fb_state_entry.E THEN
			bBusy := FALSE;
			bDone := TRUE;
		END_IF

		(*-----------------------Weiterschaltbedingungen----------------------------*)
		IF NOT bExecute AND NOT fb_state_entry.E THEN
			 bDone := FALSE;
			fb_state_entry.i16_next_step := 10;
		END_IF

(*=======================================================*)
	1000: (* Fehler *)
		IF fb_state_entry.E THEN
			bError := TRUE;
			bBusy := FALSE;
		END_IF

		(*-----------------------Weiterschaltbedingungen----------------------------*)
		IF NOT bExecute THEN
			fb_state_entry.i16_next_step := 0;
		END_IF
END_CASE

fb_state_entry(
	i16_next_step:= ,
	i16_pos:= 2,
	s_debugtext:= ,
	E=> ,
	X=> ,
	i16_step=> ,
	i16_last_step=> );
END_FUNCTION_BLOCK

(* POU EPT Lib/Funktionen/F_rSign, ST *)
FUNCTION F_rSign : LREAL
VAR_INPUT
	rValue		:LREAL;	(*Zahl*)
END_VAR
IF rValue >= 0 THEN
	F_rSign := 1;
ELSE
	F_rSign := -1;
END_IF
END_FUNCTION

(* POU EPT Lib/CamEditor/Verfahrberechnungen/ST_MFMaxMasterVelo, ST *)
FUNCTION_BLOCK ST_MFMaxMasterVelo
VAR_INPUT
	bExecute 						: BOOL;
	enu_mastertyp					: enum_ecd_typ;	(* Master ist Rund- oder Linearachse *)
	bEvCamTableChar				: BOOL;
	udiSlaveTableId					: MC_CAM_ID;	(* Slave Table-ID *)

	(* Bewegungsdaten Slave *)
	lrVeloMax						: LREAL;	(*maximale Geschwindigkeit [mm/s] an der Last/Slave *)
	lrAccMax							: LREAL;	(*maximale Beschleunigung [mm/s²] an der Last/Slave *)
	lrDecMax						: LREAL;	(*maximale Beschleunigung [mm/s²] an der Last/Slave *)

	i16_anzahl_mfps					: INT;
	lr_anfang_cam_table				: LREAL;
	lr_ende_cam_table				: LREAL;
END_VAR
VAR_OUTPUT
	bBusy							: BOOL;
	bDone							: BOOL;
	bError							: BOOL;
	udiErrorId						: UDINT;
	szErrText						: STRING;

	lrMasterVeloMax					: LREAL;
END_VAR
VAR
	stCamChar						: MC_TableCharacValues;	(*Charakteristika der Bewegungskurve*)
	fbReadCamTableCharacteristics	: MC_ReadCamTableCharacteristics;
	lrIncrement						: LREAL := 1;					(*Schrittweite Wertetabelle ACC / Integrationsschrittweite*)

	stVeloAccTable					: MC_CAM_Ref;
	aLrVeloAccData					: ARRAY[0..i_ANZAHL_PUNKTEMENGE,1..3] OF LREAL;	(*1..3  ->  MasterPos, SlaveVelo, SlaveAcc*)
	fbReadMotionFunctionValues		: MC_ReadMotionFunctionValues;
	(*===== INFO zu MotionFunktionValues: =====
	TYPE MC_ValueSelectType :
	(
	    (* a bitmask can be created by adding the following values *)
	    MC_VALUETYPE_POSITION     := 1,
	    MC_VALUETYPE_VELOCITY     := 2,
	    MC_VALUETYPE_ACCELERATION := 4,
	    MC_VALUETYPE_JERK         := 8
	);
	END_TYPE

	Mit der Auswahlmaske kann festgelegt werden, welche Daten interpoliert und zurückgeliefert werden soll.
	Der Wert entsteht durch Addition von Einzelwerten des Datentyps MC_ValueSelectType.
	Die Spaltenzahl der durch CamTable beschriebenen Datenstruktur muss der Anzahl der durch ValueSelectMask bestimmten Spaltenzahl entsprechen.
	Wenn zum Beispiel nur Positionsdaten gelesen werden, ist die Spaltenzahl 2 (Master- und Slave-Position).
	Mit jeder weiteren Ableitung (Geschwindigkeit, Beschleunigung, Ruck) kommt eine Spalte hinzu. *)

	lrMasterVelo1						: LREAL;	(*1.Mastergeschwindigkeit normiert aufgrund der max.Achsgeschwindigkeit*)
	lrMasterVelo2						: LREAL;	(*2.Reserve*)
	lrMasterVelo3						: LREAL;	(*3.Mastergeschwindigkeit normiert aufgrund der max.Achsbeschleunigung*)
	lrMasterVelo4						: LREAL;	(*4.Mastergeschwindigkeit normiert aufgrund der min.Achsbeschleunigung*)

	i								: INT;
	fb_state_entry						: ST_StateEntry;
END_VAR
VAR CONSTANT
	i_ANZAHL_PUNKTEMENGE		: INT := 360;
END_VAR
(* ======================================Schrittkette======================================== *)
fb_state_entry(
	i16_next_step:= ,
	i16_pos:= 1,
	s_debugtext:= ,
	E=> ,
	X=> ,
	i16_step=> ,
	i16_last_step=> );

CASE fb_state_entry.i16_step OF
(*=======================================================*)
	0 :	(* Init*)
		bBusy := FALSE;
		bDone := FALSE;
		bError := FALSE;
		udiErrorId := 0;
		szErrText := '';
		fbReadCamTableCharacteristics.Execute := FALSE;
		fbReadMotionFunctionValues.Execute := FALSE;
		fb_state_entry.i16_next_step := 10;

(*=======================================================*)
	10:	(* Warte Execute *)

		(*-----------------------Weiterschaltbedingungen----------------------------*)
		IF bExecute THEN
			bBusy := TRUE;
			fb_state_entry.i16_next_step := 20;
		END_IF

(*=======================================================*)
	20:	(* Prüfe Punktearray zur Anzeige der Punktewolke *)
		IF i16_anzahl_mfps > i_ANZAHL_PUNKTEMENGE THEN
			szErrText := 'Anzahl MFPs > Punktearray für Anzeige MF';
			fb_state_entry.i16_next_step := 1000;
		ELSE
			fb_state_entry.i16_next_step := 30;
		END_IF

(*=======================================================*)
	30:	(*Einlesen der Cam Table Characteristics*)
		IF fb_state_entry.E THEN
			fbReadCamTableCharacteristics.Execute := TRUE;
		END_IF

		(*-----------------------Weiterschaltbedingungen----------------------------*)
		IF fbReadCamTableCharacteristics.Busy THEN
			fb_state_entry.i16_next_step := 40;
		END_IF

(*=======================================================*)
	40:	(* Einlesen fertig  *)
		IF NOT fbReadCamTableCharacteristics.Busy THEN
			IF fbReadCamTableCharacteristics.Done THEN
				fbReadCamTableCharacteristics.Execute := FALSE;
				fb_state_entry.i16_next_step := 50;
			ELSIF fbReadCamTableCharacteristics.Error THEN
				udiErrorId := fbReadCamTableCharacteristics.ErrorID;
				szErrText := 'Fehler Einlesen charakteristische Daten';
				fb_state_entry.i16_next_step := 1000;
			END_IF
		END_IF

(*=======================================================*)
	50:	(*Geschwindigkeitsfunktion und Beschleunigungsfunktion lesen*)
		(*Upload der anzuzeigenden Punktewolke: masterPos, slaveVelo, slaveAcc mit MC_ReadMotionFunctionValues*)
		IF fb_state_entry.E THEN
			stVeloAccTable.ArraySize := SIZEOF(aLrVeloAccData);
			stVeloAccTable.pArray := ADR(aLrVeloAccData);
			stVeloAccTable.NoOfColumns := 3;	(*MasterPos, SlaveVelo, SlaveAcc*)
			stVeloAccTable.NoOfRows := i_ANZAHL_PUNKTEMENGE + 1;
			stVeloAccTable.TableType := MC_TABLETYPE_EQUIDISTANT;

			fbReadMotionFunctionValues.Execute := TRUE;
		END_IF

		(*-----------------------Weiterschaltbedingungen----------------------------*)
		IF fbReadMotionFunctionValues.Busy THEN
			fb_state_entry.i16_next_step := 60;
		END_IF

(*=======================================================*)
	60:	(* Einlesen fertig  *)
		IF NOT fbReadMotionFunctionValues.Busy THEN
			IF fbReadMotionFunctionValues.Done THEN
				fbReadMotionFunctionValues.Execute := FALSE;
				fb_state_entry.i16_next_step := 70;
			ELSIF fbReadMotionFunctionValues.Error THEN
				udiErrorId := fbReadMotionFunctionValues.ErrorID;
				szErrText := 'Beschleunigungsfunktion ungültig';
				fb_state_entry.i16_next_step := 1000;
			END_IF
		END_IF

(*=======================================================*)
	70:	(*  Berechnung der maximalen Mastergeschwindigkeit auf der Basis *)
		(*  der antriebsbedingten maximalen Geschwindigkeit des Slaves und der Tabelle.*)
		IF fb_state_entry.E THEN
			IF bEvCamTableChar THEN
				stCamChar.fSlaveVeloMin := 0;
				stCamChar.fSlaveVeloMax := 0;
				stCamChar.fSlaveAccMin := 0;
				stCamChar.fSlaveAccMax := 0;
				(* Ermittle Min- und Max-Werte für SlaveVelo und Slave Acc aus den interpolierten Daten in der Tabelle *)
				FOR i := 1 TO i_ANZAHL_PUNKTEMENGE DO
					IF aLrVeloAccData[i,2] > stCamChar.fSlaveVeloMax THEN
						stCamChar.fSlaveVeloMax := aLrVeloAccData[i,2];	(* an Position 2 -> SlaveVeloMax *)
					END_IF
					IF aLrVeloAccData[i,2] < stCamChar.fSlaveVeloMin THEN
						stCamChar.fSlaveVeloMin := aLrVeloAccData[i,2];	(* an Position 2 -> SlaveVeloMin *)
					END_IF
					IF aLrVeloAccData[i,3] > stCamChar.fSlaveAccMax THEN
						stCamChar.fSlaveAccMax := aLrVeloAccData[i,3];	(* an Position 3 -> SlaveAccMax *)
					END_IF
					IF aLrVeloAccData[i,3] < stCamChar.fSlaveAccMin THEN
						stCamChar.fSlaveAccMin := aLrVeloAccData[i,3];	(* an Position 3 -> SlaveAccMin *)
					END_IF
				END_FOR
			END_IF
		END_IF
		(*Fehlerbehandlung: Charakteristische Daten nicht konsistent*)
		(*Slave-Maximal- und Minimalgeschwindigkeit = 0*)
		IF stCamChar.fSlaveVeloMax = 0 AND stCamChar.fSlaveVeloMin = 0 THEN
			szErrText := 'Slave-Maximalgeschwindigkeit = 0';
			fb_state_entry.i16_next_step := 1000;
		(*Slave-Maximalbeschleunigung = 0*)
		ELSIF stCamChar.fSlaveAccMax = 0 THEN
			FOR i := 1 TO i_ANZAHL_PUNKTEMENGE DO
				IF aLrVeloAccData[i,3] > stCamChar.fSlaveAccMax THEN
					stCamChar.fSlaveAccMax := aLrVeloAccData[i,3];
				END_IF
			END_FOR
			IF stCamChar.fSlaveAccMax = 0 THEN
				szErrText := 'Slave-Maximalbeschleunigung = 0';
				fb_state_entry.i16_next_step := 1000;
			END_IF
		(*Slave-Minimalbeschleunigung = 0*)
		ELSIF stCamChar.fSlaveAccMin = 0 THEN
			FOR i := 1 TO i_ANZAHL_PUNKTEMENGE DO
				IF aLrVeloAccData[i,3] < stCamChar.fSlaveAccMin THEN
					stCamChar.fSlaveAccMin := aLrVeloAccData[i,3];
				END_IF
			END_FOR
			IF stCamChar.fSlaveAccMin = 0 THEN
				szErrText := 'Slave-Minimalbeschleunigung = 0';
				fb_state_entry.i16_next_step := 1000;
			END_IF
		(* Alles o.k. *)
		ELSE
			fb_state_entry.i16_next_step := 80;
		END_IF

	(*=======================================================*)
	80:	(*  Berechnung der maximalen Mastergeschwindigkeit  *)
		IF fb_state_entry.E THEN
			(* Im Kurvenscheibeneditor des Systemmanagers kann die "Normierte Darstellung" angehakt werden. *)
			(* Damit wird die Darstellung auf die maximale Achsgeschwindigkeit normiert. *)
			(*1.Mastergeschwindigkeit normiert aufgrund der max.Achsgeschwindigkeit*)
			(*Vs = Vm * Vf *)
			lrMasterVelo1 := ABS(lrVeloMax) / MAX(ABS(stCamChar.fSlaveVeloMin), ABS(stCamChar.fSlaveVeloMax));
			(*2.Reserve*)
			lrMasterVelo2 := lrMasterVelo1;
			(*3.Mastergeschwindigkeit normiert aufgrund der positiven Achsbeschleunigung*)
			(*As = Af(Sm)*Vm² + Vf(Sm)*Am *)
			lrMasterVelo3 := SQRT(ABS(MAX(lrAccMax,lrDecMax)) / ABS(stCamChar.fSlaveAccMax));
			(*4.Mastergeschwindigkeit normiert aufgrund der negativen Achsbeschleunigung*)
			(*As = Af(Sm)*Vm² + Vf(Sm)*Am *)
			lrMasterVelo4 := SQRT(ABS(MAX(lrAccMax,lrDecMax)) / ABS(stCamChar.fSlaveAccMin));
	
			lrMasterVeloMax := MIN(lrMasterVelo1, lrMasterVelo2);
			lrMasterVeloMax := MIN(lrMasterVeloMax, lrMasterVelo3);
			lrMasterVeloMax := MIN(lrMasterVeloMax, lrMasterVelo4);
		END_IF

		(*-----------------------Weiterschaltbedingungen----------------------------*)
		IF lrMasterVeloMax > 0 THEN
			fb_state_entry.i16_next_step := 90;
		ELSE
			szErrText := 'Master-Maximalbeschleunigung <= 0';
			fb_state_entry.i16_next_step := 1000;
		END_IF

(*=======================================================*)
	90: (* Fertig *)
		IF fb_state_entry.E THEN
			bBusy := FALSE;
			bDone := TRUE;
		END_IF

		(*-----------------------Weiterschaltbedingungen----------------------------*)
		IF NOT bExecute AND NOT fb_state_entry.E THEN
			 bDone := FALSE;
			fb_state_entry.i16_next_step := 10;
		END_IF

(*=======================================================*)
	1000: (* Fehler *)
		IF fb_state_entry.E THEN
			bError := TRUE;
			bBusy := FALSE;
		END_IF

		(*-----------------------Weiterschaltbedingungen----------------------------*)
		IF NOT bExecute THEN
			fb_state_entry.i16_next_step := 0;
		END_IF
END_CASE

fb_state_entry(
	i16_next_step:= ,
	i16_pos:= 2,
	s_debugtext:= ,
	E=> ,
	X=> ,
	i16_step=> ,
	i16_last_step=> );

fbReadCamTableCharacteristics(
	Execute:= ,
	CamTableID:=udiSlaveTableId,
	CamTableCharac:=stCamChar,
	Done=> ,
	Busy=> ,
	Error=> , 
	ErrorID=> );

fbReadMotionFunctionValues(
	Execute:= , 
	CamTableID:= udiSlaveTableId,
	ValueSelectMask:= MC_VALUETYPE_VELOCITY + MC_VALUETYPE_ACCELERATION,
	StartPosMaster:= lr_anfang_cam_table,
	EndPosMaster:= lr_ende_cam_table,
	Increment:= lrIncrement,
	CamTable:= stVeloAccTable,
	Done=> ,
	Busy=> , 
	Error=> ,
	ErrorID=> );
END_FUNCTION_BLOCK

(* POU EPT Lib/CamEditor/ST_Camtable_Maker, ST *)
FUNCTION_BLOCK ST_Camtable_Maker
VAR_INPUT
	st_config								: struct_config;
	st_ctrl_in								: struct_ctrl_in;

	(* Kurvenscheibendaten *)
	udiTableId							: MC_CAM_ID;			(* Table-ID *)
	arr_db_mf_tab						: ARRAY[1..i_MAX_NUM_MFP] OF struct_db_motionfunctionpoint;	(* Vorgabe aus der Datenbank *)

	lrModuloValue 						: LREAL ;
END_VAR
VAR_IN_OUT
	st_AxisRefMaster						: AXIS_REF;
	st_AxisRefSlave						: AXIS_REF;
END_VAR
VAR_OUTPUT
	st_ctrl_out							: struct_ctrl_out;
END_VAR
VAR
	st_sm						 		: struct_cameditor_meldungen;
	fb_state_entry							: ST_StateEntry;
	fb_ton_quitt							: TON;
	fb_ton_wz							: TON;

	stMotionFunctionPointDummy			: MC_MotionFunctionPoint;	(* Dummy-Punkt *)
(*	TYPE MC_MotionFunctionPoint :
		STRUCT
		    PointIndex        		: MC_MotionFunctionPoint_ID;
		    FunctionType   		: MC_MotionFunctionType;
		    PointType         		: MC_MotionPointType;
		    RelIndexNextPoint 	: MC_MotionFunctionPoint_ID;
		    MasterPos         		: LREAL; (* X *)
		    SlavePos          		: LREAL; (* Y *)
		    SlaveVelo         		: LREAL; (* Y' *)
		    SlaveAcc          		: LREAL; (* Y'' *)
		    SlaveJerk         		: LREAL; (* Y''' *)
		END_STRUCT
	END_TYPE
*)

	(*Motion Function runterschreiben an NC*)
	astWriteMotionFunction 				: ARRAY[1..i_MAX_NUM_MFP] OF MC_MotionFunctionPoint;
	stWriteMFCamTableRef				: MC_CAM_Ref;	(*Definition Zieltabelle*)
	fbCamTableSelect					: MC_CamTableSelect;
	fbWriteMF							: MC_WriteMotionFunction;
	b_cam_table_select_periodic			: BOOL := FALSE;
	b_cam_table_select_master_absolute	: BOOL := FALSE;
	b_cam_table_select_slave_absolute		: BOOL := FALSE;

	(*Motion Function hochladen von NC*)
	fbReadMF							: MC_ReadMotionFunction;
	stReadMFCamTableRef				: MC_CAM_Ref;	(*Definition Zieltabelle*)
	astReadMotionFunction 				: ARRAY[0..i_MAX_NUM_MFP] OF MC_MotionFunctionPoint;

	(*Temporäre Variablen *)
	iPointCount							: INT := 0;
	iNumMfPoints							: INT := 0;
	i_point_nr							: INT := 0;
	err_id								: UDINT := 0;
	i16_anzahl_mfps						: INT;
	lrStartPointMaster						: LREAL;	(* Startpunkt Master [°] *)
	lrStartPointSlave						: LREAL;	(* Startpunkt Slave [mm] *)
	lrEndPointMaster						: LREAL;	(* Endpunkt Master [°] *)
	lrEndPointSlave						: LREAL;	(* Endpunkt Slave [mm] *)
	lr_anfang_cam_table					: LREAL := 0;	(* Anfang Darstellungsbereich MF-Tabelle *)
	lr_ende_cam_table					: LREAL := 0;	(* Ende Darstellungsbereich MF-Tabelle *)
END_VAR
VAR CONSTANT
	i_MAX_NUM_MFP						: INT := 100;
END_VAR
fb_ton_wz(IN:= , PT:= , Q=> , ET=> );
fb_ton_quitt(IN:= , PT:= t#50ms, Q=> , ET=> );

(* ======================================Schrittkette======================================== *)
fb_state_entry(
	i16_next_step:= ,
	i16_pos:= 1,
	s_debugtext:= ,
	E=> ,
	X=> ,
	i16_step=> ,
	i16_last_step=> );

CASE fb_state_entry.i16_step OF
(*=======================================================*)
	0:	(* Init *)
		st_ctrl_out.b_bereit := FALSE;
		st_ctrl_out.b_fertig := FALSE;
		st_ctrl_out.b_fehler := FALSE;
		fbCamTableSelect.Execute := FALSE;
		fbWriteMF.Execute := FALSE;
		fbReadMF.Execute := FALSE;
		err_id := 0;
		i16_anzahl_mfps := 0;
		st_sm.lese_camtable := FALSE;
		st_sm.lese_mfp := FALSE;
		st_sm.lesen_werte_mf_tab := FALSE;
		st_sm.schreibe_camtable := FALSE;
		st_sm.schreibe_mfp := FALSE;

		fb_state_entry.i16_next_step := 10;

(*=======================================================*)
	10:	(* Warte auf Start *)
		IF lrModuloValue > 0 THEN
			b_cam_table_select_periodic := TRUE;
			b_cam_table_select_master_absolute := TRUE;
			b_cam_table_select_slave_absolute := FALSE;
		ELSE
			b_cam_table_select_periodic := FALSE;
			b_cam_table_select_master_absolute := TRUE;
			b_cam_table_select_slave_absolute := TRUE;
		END_IF

		(*-----------------------Weiterschaltbedingungen----------------------------*)
		IF st_ctrl_in.b_start THEN
			i16_anzahl_mfps := 0;
			fb_state_entry.i16_next_step := 100;
		END_IF

(*=======================================================*)
	100:	(*  *)
		IF fb_state_entry.E THEN
			FOR i_point_nr := 1 TO i_MAX_NUM_MFP BY 1 DO
				(*Für Download: Initialisieren aller  MFPs im Array *)
				astWriteMotionFunction[i_point_nr] := stMotionFunctionPointDummy;
				astWriteMotionFunction[i_point_nr].RelIndexNextPoint  := 1;

				(* Übernahme der Daten aus der WKZ-Datenbank *)
				astWriteMotionFunction[i_point_nr].FunctionType := arr_db_mf_tab[i_point_nr].FunctionType;
				astWriteMotionFunction[i_point_nr].MasterPos  := arr_db_mf_tab[i_point_nr].MasterPos;
				astWriteMotionFunction[i_point_nr].SlavePos  := arr_db_mf_tab[i_point_nr].SlavePos;
				astWriteMotionFunction[i_point_nr].PointType  := arr_db_mf_tab[i_point_nr].PointType;
				astWriteMotionFunction[i_point_nr].PointIndex  := arr_db_mf_tab[i_point_nr].PointIndex;

				IF astWriteMotionFunction[i_point_nr].FunctionType > MOTIONFUNCTYPE_NOTDEF THEN
					i16_anzahl_mfps := i16_anzahl_mfps + 1;
				END_IF
			END_FOR

			(* Beim Letzen Punkt in der Tabelle immer den RelIndexNextPoint auf 0 setzen *)
			astWriteMotionFunction[i16_anzahl_mfps].RelIndexNextPoint := 0;

			(* Darstellungsbereich der MF-Tabelle (wird benötigt für die Funktion "MC_ReadMotionFunctionValues") *)
			IF lrModuloValue > 0 THEN
				lr_anfang_cam_table := 0;
				lr_ende_cam_table := lrModuloValue;
			ELSE
				lr_anfang_cam_table := arr_db_mf_tab[1].MasterPos;
				lr_ende_cam_table := arr_db_mf_tab[i16_anzahl_mfps].MasterPos;
			END_IF
		END_IF

		(*-----------------------Weiterschaltbedingungen----------------------------*)
		fb_state_entry.i16_next_step := 110;

(*=======================================================*)
	110:	(* Alle Punkte der MF-Tabelle werden an die NC runter geschrieben  *)
		IF fb_state_entry.E THEN
			iNumMfPoints := i16_anzahl_mfps;
			(*Tabelle initialisieren *)
			stWriteMFCamTableRef.pArray := ADR(astWriteMotionFunction[1]);	(* Adresse des ersten eindimensionalen Arrays vom Typ MC_MotionFunctionPoint. Jedes Array-Element enthält eine Beschreibung einer Stützstelle der Kurvenscheibe. *)
			stWriteMFCamTableRef.ArraySize := SIZEOF(astWriteMotionFunction[1]) * iNumMfPoints;
			stWriteMFCamTableRef.TableType := MC_TABLETYPE_MOTIONFUNCTION;
			stWriteMFCamTableRef.NoOfColumns := 1;	(* Bei Table Type "MC_TABLETYPE_MOTIONFUNCTION" ist NoOfColumns immer 1 *)
			stWriteMFCamTableRef.NoOfRows := iNumMfPoints;

			fbCamTableSelect.Execute := TRUE;
		END_IF

		(*-----------------------Weiterschaltbedingungen----------------------------*)
		IF fbCamTableSelect.Busy THEN
			fb_state_entry.i16_next_step := 120;
		END_IF

(*=======================================================*)
	120:	(* Alle Punkte der MF-Tabelle werden an die NC runter geschrieben  *)
		IF NOT fbCamTableSelect.Busy THEN
			IF fbCamTableSelect.Done THEN
				fbCamTableSelect.Execute := FALSE;
				fb_state_entry.i16_next_step := 200;
			ELSIF fbCamTableSelect.Error THEN
				st_sm.schreibe_camtable := TRUE;
				err_id := fbCamTableSelect.ErrorID;
				fb_state_entry.i16_next_step := 1000;
			END_IF
		END_IF

(*=======================================================*)
	200:	(* Lesen der MF-Tabelle von der NC  *)
		IF fb_state_entry.E THEN
			stReadMFCamTableRef.pArray := ADR(astReadMotionFunction[0]);
			stReadMFCamTableRef.ArraySize := SIZEOF(astReadMotionFunction[0]) * (iNumMfPoints + 1) ;
			stReadMFCamTableRef.NoOfColumns := 2;		(* Master und Slave Spalte*)
			stReadMFCamTableRef.NoOfRows := iNumMfPoints;
			stReadMFCamTableRef.TableType := MC_TABLETYPE_MOTIONFUNCTION;
			
			(* Für Upload initialisieren *)
			FOR iPointCount := 1 TO i_MAX_NUM_MFP DO
				astReadMotionFunction[iPointCount] := stMotionFunctionPointDummy;
			END_FOR

			fbReadMF.Execute := TRUE;
		END_IF

		(*-----------------------Weiterschaltbedingungen----------------------------*)
		IF fbReadMF.Busy THEN
			fb_state_entry.i16_next_step := 210;
		END_IF

(*=======================================================*)
	210:	(* Die gesamte MF-Tabelle hochladen  *)
		IF NOT fbReadMF.Busy THEN
			IF fbReadMF.Done THEN
				fbReadMF.Execute := FALSE;
				fb_state_entry.i16_next_step := 220;
			ELSIF fbReadMF.Error THEN
				st_sm.lese_camtable := TRUE;
				err_id := fbReadMF.ErrorID;
				fb_state_entry.i16_next_step := 1000;
			END_IF
		END_IF

(*=======================================================*)
	220:	(* Fertig  *)
		IF fb_state_entry.E THEN
			st_ctrl_out.b_fertig := TRUE;
		END_IF

		(*-----------------------Weiterschaltbedingungen----------------------------*)
		IF NOT st_ctrl_in.b_start THEN
			st_ctrl_out.b_fertig := FALSE;
			fb_state_entry.i16_next_step := 10;
		END_IF

(*=======================================================*)
	FEHLER: (* Fehler *)
		IF fb_state_entry.E THEN
			st_ctrl_out.b_fehler := TRUE;
			fb_ton_quitt.IN := FALSE;
		END_IF

		(*-----------------------Weiterschaltbedingungen----------------------------*)
		IF st_ctrl_in.b_quitt AND NOT fb_state_entry.E THEN
			st_ctrl_out.b_fehler := FALSE;
			fb_ton_quitt.IN := TRUE;
		END_IF

		IF fb_ton_quitt.Q THEN
			fb_ton_quitt.IN := FALSE;
			fb_state_entry.i16_next_step := 0;
		END_IF
END_CASE

fb_state_entry(
	i16_next_step:= ,
	i16_pos:= 2,
	s_debugtext:= ,
	E=> ,
	X=> ,
	i16_step=> ,
	i16_last_step=> );

(* Erstellen einer neuen MF-Tabelle mit anschliessendem Füllen der Punktdaten: *)
(* Es wird eine neue Tabelle in der NC angelegt zudem werden  Master und Slave Achsen zugeordnet. *)
(* Die Länge der Tabelle mit ihren Punktdaten wird gleichzeitig mit reingeschrieben. *)
fbCamTableSelect(
	Execute:= , 
	Periodic:= b_cam_table_select_periodic,
	MasterAbsolute:= b_cam_table_select_master_absolute,
	SlaveAbsolute:= b_cam_table_select_slave_absolute,
	CamTableID:= udiTableId,
	Master := st_AxisRefMaster,
	Slave := st_AxisRefSlave,
	CamTable:= stWriteMFCamTableRef,
	Done=> ,
	Busy=> , 
	Error=> , 
	ErrorID=> );

(* Die gesamte Tabelle einlesen aus der NC *)
fbReadMF(
	Execute:= ,
	CamTableID:= udiTableId,
	PointID:= 1,
	NumPoints:= stReadMFCamTableRef.NoOfRows,
	CamTable:= stReadMFCamTableRef,
	Done=> ,
	Busy=> ,
	Error=> ,
	ErrorID=> ,
	NumPointsRead=> );

(* Die ganze MF-Tabelle schreiben *)
fbWriteMF(
	Execute:= ,
	CamTableID:= udiTableId,
	PointID:= 1,
	NumPoints:= i16_anzahl_mfps,
	CamTable:= stWriteMFCamTableRef,
	Done=> ,
	Busy=> , 
	Error=> , 
	ErrorID=> );

IF st_config.b_config_fertig THEN
	garr_stoermeldungen[st_config.i16_meld_startindex + 0] := st_sm.lese_mfp;
	garr_stoermeldungen[st_config.i16_meld_startindex + 1] := st_sm.lese_camtable;
	garr_stoermeldungen[st_config.i16_meld_startindex + 2] := st_sm.lesen_werte_mf_tab;
	garr_stoermeldungen[st_config.i16_meld_startindex + 3] := st_sm.schreibe_mfp;
	garr_stoermeldungen[st_config.i16_meld_startindex + 4] := st_sm.schreibe_camtable;
	garr_stoermeldungen[st_config.i16_meld_startindex + 5] := FALSE;
	garr_stoermeldungen[st_config.i16_meld_startindex + 6] := FALSE;
	garr_stoermeldungen[st_config.i16_meld_startindex + 7] := FALSE;
	garr_stoermeldungen[st_config.i16_meld_startindex + 8] := FALSE;
	garr_stoermeldungen[st_config.i16_meld_startindex + 9] := FALSE;
	garr_stoermeldungen[st_config.i16_meld_startindex + 10] := FALSE;
	garr_stoermeldungen[st_config.i16_meld_startindex + 11] := FALSE;
	garr_stoermeldungen[st_config.i16_meld_startindex + 12] := FALSE;
	garr_stoermeldungen[st_config.i16_meld_startindex + 13] := FALSE;
	garr_stoermeldungen[st_config.i16_meld_startindex + 14] := FALSE;
	garr_stoermeldungen[st_config.i16_meld_startindex + 15] := FALSE;
	garr_stoermeldungen[st_config.i16_meld_startindex + 16] := FALSE;
	garr_stoermeldungen[st_config.i16_meld_startindex + 17] := FALSE;
	garr_stoermeldungen[st_config.i16_meld_startindex + 18] := FALSE;
	garr_stoermeldungen[st_config.i16_meld_startindex + 19] := FALSE;
	
	garr_betriebsmeldungen[st_config.i16_meld_startindex + 0] := FALSE;
	garr_betriebsmeldungen[st_config.i16_meld_startindex + 1] := FALSE;
	garr_betriebsmeldungen[st_config.i16_meld_startindex + 2] := FALSE;
	garr_betriebsmeldungen[st_config.i16_meld_startindex + 3] := FALSE;
	garr_betriebsmeldungen[st_config.i16_meld_startindex + 4] := FALSE;
	garr_betriebsmeldungen[st_config.i16_meld_startindex + 5] := FALSE;
	garr_betriebsmeldungen[st_config.i16_meld_startindex + 6] := FALSE;
	garr_betriebsmeldungen[st_config.i16_meld_startindex + 7] := FALSE;
	garr_betriebsmeldungen[st_config.i16_meld_startindex + 8] := FALSE;
	garr_betriebsmeldungen[st_config.i16_meld_startindex + 9] := FALSE;
	garr_betriebsmeldungen[st_config.i16_meld_startindex + 10] := FALSE;
	garr_betriebsmeldungen[st_config.i16_meld_startindex + 11] := FALSE;
	garr_betriebsmeldungen[st_config.i16_meld_startindex + 12] := FALSE;
	garr_betriebsmeldungen[st_config.i16_meld_startindex + 13] := FALSE;
	garr_betriebsmeldungen[st_config.i16_meld_startindex + 14] := FALSE;
	garr_betriebsmeldungen[st_config.i16_meld_startindex + 15] := FALSE;
	garr_betriebsmeldungen[st_config.i16_meld_startindex + 16] := FALSE;
	garr_betriebsmeldungen[st_config.i16_meld_startindex + 17] := FALSE;
	garr_betriebsmeldungen[st_config.i16_meld_startindex + 18] := FALSE;
	garr_betriebsmeldungen[st_config.i16_meld_startindex + 19] := FALSE;
END_IF
END_FUNCTION_BLOCK

(* POU EPT Lib/CamEditor/ST_Kurvenscheibeneditor, ST *)
FUNCTION_BLOCK ST_Kurvenscheibeneditor
VAR_INPUT
 	udint_camtable_id						: UDINT;
	i16_laenge_mfp_tabelle				: UINT;
	arr_db_mfps							: ARRAY[1..ui_MAX_NUM_MFP] OF struct_db_motionfunctionpoint;	(* Vorgabe aus der Datenbank *)
	st_config								: struct_config;
	st_ctrl_in								: struct_ctrl_in;
END_VAR
VAR_IN_OUT
	i16_auftrag							: enum_auftrag_cameditor;
END_VAR
VAR_OUTPUT
	st_ctrl_out							: struct_ctrl_out;
END_VAR
VAR
	mc_point_id							: MC_MotionFunctionPoint_ID;
	mc_read_motion_function_point			: MC_ReadMotionFunctionPoint;
	mc_write_motion_function_point			: MC_WriteMotionFunctionPoint;
	arr_motion_function_points				: ARRAY[1..ui_MAX_NUM_MFP] OF MC_MotionFunctionPoint;	(* Eingelesene Kurvenscheibentabelle aus dem Systemmanager oder geschriebene MFPs an den Systemmanager *)
	udint_write_error_id 					: UDINT := 0;
	udint_read_error_id					: UDINT := 0;
	fb_state_entry							: ST_StateEntry;
	fb_ton_quitt							: TON;
	fb_ton_wz							: TON;
	fb_r_trig_ibn_lesen					: R_TRIG;
	fb_r_trig_ibn_schreiben					: R_TRIG;
	fb_ton_ibn_lesen						: TON;
	fb_ton_ibn_schreiben					: TON;
	b_ibn_lesen							: BOOL := FALSE;
	b_ibn_schreiben						: BOOL := FALSE;
	sm_fehler_schreibe_mfp 				: BOOL := FALSE;
	sm_fehler_lese_mfp					: BOOL := FALSE;
END_VAR
VAR CONSTANT
	ui_MAX_NUM_MFP					:UINT := 100;
END_VAR
fb_ton_wz(IN:= , PT:= , Q=> , ET=> );
fb_ton_quitt(IN:= , PT:= t#100ms, Q=> , ET=> );

fb_r_trig_ibn_lesen(CLK:= b_ibn_lesen, Q=> );
fb_r_trig_ibn_schreiben(CLK:= b_ibn_schreiben, Q=> );
fb_ton_ibn_lesen(IN:= , PT:= t#1s, Q=> , ET=> );
fb_ton_ibn_schreiben(IN:= , PT:= t#1s, Q=> , ET=> );


IF fb_r_trig_ibn_lesen.Q THEN
	fb_ton_ibn_lesen.IN := TRUE;
ELSE
	IF fb_ton_ibn_lesen.Q THEN
		b_ibn_lesen := FALSE;
	 	fb_ton_ibn_lesen.IN := FALSE;
	END_IF
END_IF

IF fb_r_trig_ibn_schreiben.Q THEN
	fb_ton_ibn_schreiben.IN := TRUE;
ELSE
	IF fb_ton_ibn_schreiben.Q THEN
		b_ibn_schreiben := FALSE;
	 	fb_ton_ibn_schreiben.IN := FALSE;
	END_IF
END_IF

(* ======================================Schrittkette======================================== *)
fb_state_entry(
	i16_next_step:= ,
	i16_pos:= 1,
	s_debugtext:= ,
	E=> ,
	X=> ,
	i16_step=> ,
	i16_last_step=> );

CASE fb_state_entry.i16_step OF
(*=======================================================*)
	0:	(* Init *)
		fb_ton_quitt.IN := FALSE;
		st_ctrl_out.b_bereit := FALSE;
		st_ctrl_out.b_fehler := FALSE;
		i16_auftrag := MFP_KEIN_AUFTRAG;
		mc_point_id := 1;
		mc_read_motion_function_point.Execute := FALSE;
		mc_write_motion_function_point.Execute := FALSE;
		sm_fehler_schreibe_mfp := FALSE;
		sm_fehler_lese_mfp := FALSE;
		fb_state_entry.i16_next_step := 10;

(*=======================================================*)
	10: (* Warte auf Auftrag *)
		IF fb_state_entry.E THEN
			st_ctrl_out.b_bereit := TRUE;
		END_IF

		(* Motion Function Points aus der Kurvenscheibentabelle des Systemmanagers lesen *)
		IF i16_auftrag = MFP_LESEN OR fb_r_trig_ibn_lesen.Q THEN
			fb_state_entry.i16_next_step := 100;
		(* Motion Function Points von der Datenbankvorgabe in die Kurvenscheibentabelle des Systemmanagers schreiben *)
		ELSIF i16_auftrag = MFP_SCHREIBEN OR fb_r_trig_ibn_schreiben.Q THEN
			fb_state_entry.i16_next_step := 200;
		END_IF

(*=======================================================*)
	100:
		mc_point_id := 1;
		fb_state_entry.i16_next_step := 110;

(*=======================================================*)
	110:	(* Lese die einzelnen MFPs aus der Kurvenscheibentabelle des Systemmanagers *)
		IF fb_state_entry.E THEN
			mc_read_motion_function_point.Execute := TRUE;
		END_IF

		IF mc_read_motion_function_point.Busy THEN
			mc_read_motion_function_point.Execute := FALSE;
			fb_state_entry.i16_next_step := 120;
		END_IF

(*=======================================================*)
	120:	(* MFP wurde gelesen *)
		IF  NOT mc_read_motion_function_point.Busy THEN
			IF NOT mc_read_motion_function_point.Error THEN
				fb_state_entry.i16_next_step := 130;
			ELSE
				sm_fehler_schreibe_mfp := TRUE;
				fb_state_entry.i16_next_step := FEHLER;
			END_IF
		END_IF

(*=======================================================*)
	130:	(* Zum nächsten MFP *)
		IF fb_state_entry.E THEN
			mc_point_id := mc_point_id + 1;
		END_IF

		IF mc_point_id > i16_laenge_mfp_tabelle THEN
			(* Alle Punkte wurden gelesen *)
			fb_state_entry.i16_next_step := 140;
		ELSE
			(* Weitere Punkte lesen *)
			fb_state_entry.i16_next_step := 110;
		END_IF

(*=======================================================*)
	140:	(* Lesevorgang beendet *)
		fb_state_entry.i16_next_step := 0;

(*=======================================================*)
	200:	(* Einlesen der Vorgabepunktetabelle *)
		IF fb_state_entry.E THEN
			FOR mc_point_id := 1  TO 32 BY 1DO
				arr_motion_function_points[mc_point_id].PointIndex := arr_db_mfps[mc_point_id].PointIndex;
				arr_motion_function_points[mc_point_id].FunctionType := arr_db_mfps[mc_point_id].FunctionType;
				arr_motion_function_points[mc_point_id].PointType := arr_db_mfps[mc_point_id].PointType;
				arr_motion_function_points[mc_point_id].RelIndexNextPoint := 1;
				arr_motion_function_points[mc_point_id].MasterPos := arr_db_mfps[mc_point_id].MasterPos;
				arr_motion_function_points[mc_point_id].SlavePos := arr_db_mfps[mc_point_id].SlavePos;
			END_FOR
		END_IF
		mc_point_id := 1;
		fb_state_entry.i16_next_step := 210;

(*=======================================================*)
	210:	(* Schreibe die einzelnen MFPs *)
		IF fb_state_entry.E THEN
			mc_write_motion_function_point.Execute := TRUE;
		END_IF

		IF mc_write_motion_function_point.Busy THEN
			mc_write_motion_function_point.Execute := FALSE;
			fb_state_entry.i16_next_step := 220;
		END_IF

(*=======================================================*)
	220:	(* MFP wurde geschrieben *)
		IF  NOT mc_write_motion_function_point.Busy THEN
			IF NOT  mc_write_motion_function_point.Error THEN
				fb_state_entry.i16_next_step := 230;
			ELSE
				sm_fehler_schreibe_mfp := TRUE;
				fb_state_entry.i16_next_step := FEHLER;
			END_IF
		END_IF

(*=======================================================*)
	230:	(* Zum nächsten MFP *)
		IF fb_state_entry.E THEN
			mc_point_id := mc_point_id + 1;
		END_IF

		IF mc_point_id > i16_laenge_mfp_tabelle THEN
			(* Alle Punkte wurden gelesen *)
			fb_state_entry.i16_next_step := 240;
		ELSE
			(* Weitere Punkte lesen *)
			fb_state_entry.i16_next_step := 210;
		END_IF

(*=======================================================*)
	240:	(* Schreibevorgang beendet *)
		fb_state_entry.i16_next_step := 0;

(*=======================================================*)
	1000: (* Fehler *)
		IF fb_state_entry.E THEN
			st_ctrl_out.b_fehler := TRUE;
			fb_ton_quitt.IN := FALSE;
		END_IF

		(*-----------------------Weiterschaltbedingungen----------------------------*)
		IF st_ctrl_in.b_quitt AND NOT fb_state_entry.E THEN
			st_ctrl_out.b_fehler := FALSE;
			fb_ton_quitt.IN := TRUE;
		END_IF

		IF fb_ton_quitt.Q THEN
			fb_ton_quitt.IN := FALSE;
			fb_state_entry.i16_next_step := 0;
		END_IF
END_CASE

fb_state_entry(
	i16_next_step:= ,
	i16_pos:= 2,
	s_debugtext:= ,
	E=> ,
	X=> ,
	i16_step=> ,
	i16_last_step=> );

mc_read_motion_function_point(
	Execute:= ,
	CamTableID:= udint_camtable_id,
	PointID:= mc_point_id,
	Point:= arr_motion_function_points[mc_point_id],
	Done=> , 
	Busy=> , 
	Error=> , 
	ErrorID=> );

mc_write_motion_function_point(
	Execute:= , 
	CamTableID:= udint_camtable_id,
	PointID:= mc_point_id,
	Point:= arr_motion_function_points[mc_point_id],
	Done=> , 
	Busy=> , 
	Error=> , 
	ErrorID=> );

IF st_config.b_config_fertig THEN
	garr_stoermeldungen[st_config.i16_meld_startindex + 0] := sm_fehler_lese_mfp;
	garr_stoermeldungen[st_config.i16_meld_startindex + 1] := sm_fehler_schreibe_mfp;
	garr_stoermeldungen[st_config.i16_meld_startindex + 2] := FALSE;
	garr_stoermeldungen[st_config.i16_meld_startindex + 3] := FALSE;
	garr_stoermeldungen[st_config.i16_meld_startindex + 4] := FALSE;
	garr_stoermeldungen[st_config.i16_meld_startindex + 5] := FALSE;
	garr_stoermeldungen[st_config.i16_meld_startindex + 6] := FALSE;
	garr_stoermeldungen[st_config.i16_meld_startindex + 7] := FALSE;
	garr_stoermeldungen[st_config.i16_meld_startindex + 8] := FALSE;
	garr_stoermeldungen[st_config.i16_meld_startindex + 9] := FALSE;
	garr_stoermeldungen[st_config.i16_meld_startindex + 10] := FALSE;
	garr_stoermeldungen[st_config.i16_meld_startindex + 11] := FALSE;
	garr_stoermeldungen[st_config.i16_meld_startindex + 12] := FALSE;
	garr_stoermeldungen[st_config.i16_meld_startindex + 13] := FALSE;
	garr_stoermeldungen[st_config.i16_meld_startindex + 14] := FALSE;
	garr_stoermeldungen[st_config.i16_meld_startindex + 15] := FALSE;
	garr_stoermeldungen[st_config.i16_meld_startindex + 16] := FALSE;
	garr_stoermeldungen[st_config.i16_meld_startindex + 17] := FALSE;
	garr_stoermeldungen[st_config.i16_meld_startindex + 18] := FALSE;
	garr_stoermeldungen[st_config.i16_meld_startindex + 19] := FALSE;
	
	garr_betriebsmeldungen[st_config.i16_meld_startindex + 0] := FALSE;
	garr_betriebsmeldungen[st_config.i16_meld_startindex + 1] := FALSE;
	garr_betriebsmeldungen[st_config.i16_meld_startindex + 2] := FALSE;
	garr_betriebsmeldungen[st_config.i16_meld_startindex + 3] := FALSE;
	garr_betriebsmeldungen[st_config.i16_meld_startindex + 4] := FALSE;
	garr_betriebsmeldungen[st_config.i16_meld_startindex + 5] := FALSE;
	garr_betriebsmeldungen[st_config.i16_meld_startindex + 6] := FALSE;
	garr_betriebsmeldungen[st_config.i16_meld_startindex + 7] := FALSE;
	garr_betriebsmeldungen[st_config.i16_meld_startindex + 8] := FALSE;
	garr_betriebsmeldungen[st_config.i16_meld_startindex + 9] := FALSE;
	garr_betriebsmeldungen[st_config.i16_meld_startindex + 10] := FALSE;
	garr_betriebsmeldungen[st_config.i16_meld_startindex + 11] := FALSE;
	garr_betriebsmeldungen[st_config.i16_meld_startindex + 12] := FALSE;
	garr_betriebsmeldungen[st_config.i16_meld_startindex + 13] := FALSE;
	garr_betriebsmeldungen[st_config.i16_meld_startindex + 14] := FALSE;
	garr_betriebsmeldungen[st_config.i16_meld_startindex + 15] := FALSE;
	garr_betriebsmeldungen[st_config.i16_meld_startindex + 16] := FALSE;
	garr_betriebsmeldungen[st_config.i16_meld_startindex + 17] := FALSE;
	garr_betriebsmeldungen[st_config.i16_meld_startindex + 18] := FALSE;
	garr_betriebsmeldungen[st_config.i16_meld_startindex + 19] := FALSE;
END_IF
END_FUNCTION_BLOCK

(* POU EPT Lib/Ethercat Diagnose/FB_EtherCatDiag, ST *)
FUNCTION_BLOCK FB_EtherCatDiag
VAR_INPUT
	st_config					: struct_config;
	st_ctrl_in					: struct_ctrl_in;
END_VAR
VAR_OUTPUT
	st_ctrl_out						: struct_ctrl_out;
END_VAR
VAR
	fb_state_entry					: ST_StateEntry;
	visu_Data						: struct_EthercatDiagnose;
	fb_ton_start						: TON;
	fb_ton_quitt						: TON;
	FB_EcGetAllSlaveStates			: FB_EcGetAllSlaveStates;
	by_AmsNetId					AT %I* : T_AmsNetIdArr;			(*Muss verknüpft werden*)
	s_AmsNetId					: T_AmsNetId := '0.0.0.0.0.0';	(* Master ID*)
	st_EcSlaveStateData			: ARRAY[1..MaxNoOfSlaves] OF ST_EcSlaveState;
	i_Slaves						: INT; 						(* Anzahl konfigurierter Slaves*)
	i								: INT;
	nErrId							: UDINT;

	sm_FehlerEthercat				: BOOL;

	FB_EcGetConfSlaves			: FB_EcGetConfSlaves;
	st_EcGetConfSlavesData		: ARRAY[1..MaxNoOfSlaves] OF ST_EcSlaveConfigData;


	fb_EcMasterFrameStatistic		: FB_EcMasterFrameStatistic;
END_VAR
(*======================================================
   ST: Fb_EtherCatDiag
 ------------------------------------------------------
   Auth: 	Thomas Vilgis, Werner Friedl    						 
   Date: 	25.01.2019    						     
   Rev.: 		1.1	
   Desc:		1.0	
				Der Baustein liest alle Zustände der Slaves aus.
   				Es muss nur die Variable "by_AmsNetId" mit dem EtherCAT Master verknüpt werden.
				Die maximale Anzahl an Slaves wird durch die globale Konstante "MaxNoOfSlaves" begrenzt.
				In der Visu werden die ausgelesenen Daten wie im Systemmanager angezeigt.
				Es wird eine Fehlermeldung ausgegeben, dass mindestens ein Teilnehmer nicht OP ist.
				Dies wird aber nur gemacht, wenn "st_config.b_station_aktiv" TRUE ist.
			1.1 
				UP und Down Button entfernt
				Var visu_Data.st_Slave[1].b_Err hinzugefüt => damit werden in der Visu Zeilen im Fehler farbig dargestellt.
			
   Historie: 	1.0

 ========================================================*)

(* Zeiten *)
fb_ton_start(IN:= NOT fb_ton_start.Q, PT:= T#2s, Q=>  , ET=> );
fb_ton_quitt(IN:= , PT:= t#100ms, Q=> , ET=> );
(* Flanken *)

(* ======================================Schrittkette======================================== *)
fb_state_entry(i16_pos:= 1);

CASE fb_state_entry.i16_step OF
(*=======================================================*)
	INIT_OBJ:	(*initialisieren*)

		(*-----------------------Weiterschaltbedingungen----------------------------*)
		IF st_config.b_config_fertig THEN
			fb_state_entry.i16_next_step:=INIT;
		END_IF
		
(*=======================================================*)
	INIT:	(*initialisieren*)
		IF fb_state_entry.E THEN
			fb_EcGetAllSlaveStates.bExecute := FALSE;
			fb_EcGetConfSlaves.bExecute := FALSE;
			fb_EcMasterFrameStatistic.bExecute := FALSE;
			sm_FehlerEthercat := FALSE;

			(*Umwandeln in einen String*)
			s_AmsNetId := F_CreateAmsNetId(by_AmsNetId);
		END_IF

		(*-----------------------Weiterschaltbedingungen----------------------------*)
		IF s_AmsNetId <> '0.0.0.0.0.0' THEN
			fb_state_entry.i16_next_step:=20;
		END_IF

(*=======================================================*)
	20:(* Baustein zum Abfragen der Configuration starten*)
		IF fb_state_entry.E THEN
			fb_EcGetConfSlaves.bExecute:=TRUE;
		END_IF

		(*-----------------------Weiterschaltbedingungen----------------------------*)
		IF 	fb_EcGetConfSlaves.bBusy THEN
			fb_state_entry.i16_next_step:=30;
		END_IF

(*=======================================================*)
	30:(* Warte auf Baustein *)

		(*-----------------------Weiterschaltbedingungen----------------------------*)
		IF NOT fb_EcGetConfSlaves.bBusy THEN
			fb_EcGetConfSlaves.bExecute:=FALSE;
			IF 	fb_EcGetConfSlaves.bError THEN
				nErrId:=fb_EcGetConfSlaves.nErrorId;
				fb_state_entry.i16_next_step:=FEHLER;
			ELSE
				fb_state_entry.i16_next_step:=BEREIT;
			END_IF
		END_IF
		
(*=======================================================*)
	BEREIT:	(*  *)
		IF fb_state_entry.E THEN
			LeseDaten();
		END_IF

		(*-----------------------Weiterschaltbedingungen----------------------------*)
		IF fb_ton_start.Q THEN
			fb_state_entry.i16_next_step:=110;
		END_IF

(*=======================================================*)
	110:(* Baustein zum Abfragen des Status starten*)
		IF fb_state_entry.E THEN
			fb_EcGetAllSlaveStates.bExecute:=TRUE;
		END_IF

		(*-----------------------Weiterschaltbedingungen----------------------------*)
		IF 	fb_EcGetAllSlaveStates.bBusy THEN
			fb_state_entry.i16_next_step:=120;
		END_IF

(*=======================================================*)
	120:(* Warte auf Baustein *)

		(*-----------------------Weiterschaltbedingungen----------------------------*)
		IF NOT fb_EcGetAllSlaveStates.bBusy THEN
			fb_EcGetAllSlaveStates.bExecute:=FALSE;
			IF 	fb_EcGetAllSlaveStates.bError THEN
				nErrId:=fb_EcGetAllSlaveStates.nErrId;
				fb_state_entry.i16_next_step:=FEHLER;
			ELSE
				i_Slaves := UINT_TO_INT(fb_EcGetAllSlaveStates.nSlaves);
				fb_state_entry.i16_next_step:=130;
			END_IF
		END_IF

(*=======================================================*)
	130:(* Prüfe, ob ein Slave einen Fehler hat *)
		IF fb_state_entry.E THEN
			sm_FehlerEthercat := FALSE;
			(*Fehlermeldung nur ausgeben, wenn Sation aktiv ist*)
			IF st_config.b_station_aktiv THEN
				FOR i:= 1 TO i_Slaves DO
					IF st_EcSlaveStateData[i].deviceState <> EC_DEVICE_STATE_OP THEN
						visu_Data.st_Slave[i].b_Err:=TRUE;
						sm_FehlerEthercat := TRUE;
						(*-----------------------Weiterschaltbedingungen----------------------------*)
						fb_state_entry.i16_next_step:=FEHLER;
					ELSE
						visu_Data.st_Slave[i].b_Err:=FALSE;
						(*-----------------------Weiterschaltbedingungen----------------------------*)
						fb_state_entry.i16_next_step:=140;
					END_IF
				END_FOR
			END_IF
		END_IF

(*=======================================================*)
	140:(* Baustein zum Abfragen der Lost Frames starten*)
		IF fb_state_entry.E THEN
			fb_EcMasterFrameStatistic.bExecute:=TRUE;
		END_IF

		(*-----------------------Weiterschaltbedingungen----------------------------*)
		IF 	fb_EcMasterFrameStatistic.bBusy THEN
			fb_state_entry.i16_next_step:=150;
		END_IF

(*=======================================================*)
	150:(* Warte auf Baustein *)

		(*-----------------------Weiterschaltbedingungen----------------------------*)
		IF NOT fb_EcMasterFrameStatistic.bBusy THEN
			fb_EcMasterFrameStatistic.bExecute:=FALSE;
			IF 	fb_EcMasterFrameStatistic.bError THEN
				nErrId:=fb_EcMasterFrameStatistic.nErrId;
				fb_state_entry.i16_next_step:=FEHLER;
			ELSE
				fb_state_entry.i16_next_step:=BEREIT;
			END_IF
		END_IF



(*=======================================================*)
	FEHLER:
		IF fb_state_entry.E THEN
			fb_ton_quitt.IN := FALSE;
			st_ctrl_out.b_fehler := TRUE;
		END_IF

		(*-----------------------Weiterschaltbedingungen----------------------------*)
		IF st_ctrl_in.b_quitt AND NOT fb_state_entry.E THEN
			st_ctrl_out.b_fehler := FALSE;
			fb_ton_quitt.IN := TRUE;
		END_IF

		IF fb_ton_quitt.Q THEN
			fb_ton_quitt.IN := FALSE;
			fb_state_entry.i16_next_step := INIT;
		END_IF

END_CASE


fb_state_entry(i16_pos:= 2);


(*Aufruf*)
fb_EcGetAllSlaveStates(
	sNetId:= s_AmsNetId, 
	pStateBuf:= ADR(st_EcSlaveStateData),
	cbBufLen:= SIZEOF(st_EcSlaveStateData));

fb_EcGetConfSlaves(
	sNetId:= s_AmsNetId,
	pArrEcConfSlaveInfo:= ADR(st_EcGetConfSlavesData),
	cbBufLen:= SIZEOF(st_EcGetConfSlavesData) );

fb_EcMasterFrameStatistic(
	sNetId:= s_AmsNetId);
	


IF st_config.b_config_fertig THEN
	(* Fehlermeldungen und Betriebsmeldungen ab dem Startindex in die globalen Meldungsarrays schreiben *)
	garr_stoermeldungen[st_config.i16_meld_startindex + 0] := sm_FehlerEthercat;
	garr_stoermeldungen[st_config.i16_meld_startindex + 1] := FALSE;
	garr_stoermeldungen[st_config.i16_meld_startindex + 2] := FALSE;
	garr_stoermeldungen[st_config.i16_meld_startindex + 3] := FALSE;
	garr_stoermeldungen[st_config.i16_meld_startindex + 4] := FALSE;

	garr_betriebsmeldungen[st_config.i16_meld_startindex + 0] := FALSE;
	garr_betriebsmeldungen[st_config.i16_meld_startindex + 1] := FALSE;
	garr_betriebsmeldungen[st_config.i16_meld_startindex + 2] := FALSE;
	garr_betriebsmeldungen[st_config.i16_meld_startindex + 3] := FALSE;
	garr_betriebsmeldungen[st_config.i16_meld_startindex + 4] := FALSE;
END_IF
END_FUNCTION_BLOCK
ACTION LeseDaten:
(*Master Daten übergeben*)
visu_Data.ST_Master.s_Name := st_config.str_instanz_name;
visu_Data.st_Master.s_AmsNetId := s_AmsNetId;
visu_Data.st_Master.i_Slaves := i_Slaves;
visu_Data.st_Master.f_FramesPerSeconed := fb_EcMasterFrameStatistic.fFramesPerSecond;
visu_Data.st_Master.i_LostFrames := fb_EcMasterFrameStatistic.nLostFrames;

(*Slave Daten übergeben*)
FOR i:=1 TO MaxNoOfSlaves DO
	visu_Data.st_Slave[i].i_Number := i;
	IF st_EcGetConfSlavesData[i].nAddr <> 0 THEN
		visu_Data.st_Slave[i].s_Adress := WORD_TO_STRING(st_EcGetConfSlavesData[i].nAddr);
	END_IF
	visu_Data.st_Slave[i].s_Name := st_EcGetConfSlavesData[i].sName;
	visu_Data.st_Slave[i].s_Type := st_EcGetConfSlavesData[i].sType;

	visu_Data.st_Slave[i].s_DeviceState := F_ConvStateToString(st_EcSlaveStateData[i].deviceState);

	(*Link State wird von TwinCAT aus Status und Port-Nummer zusammengebaut*)
	CASE st_EcSlaveStateData[i].linkState OF
		0:
			;	(*alles OK*)
		1:
			visu_Data.st_Slave[i].s_DeviceState := CONCAT(visu_Data.st_Slave[i].s_DeviceState, ' NO_COMM');
			
		18:
			visu_Data.st_Slave[i].s_DeviceState := CONCAT(visu_Data.st_Slave[i].s_DeviceState, ' LINK_WITHOUT_COMM A');
		34:
			visu_Data.st_Slave[i].s_DeviceState := CONCAT(visu_Data.st_Slave[i].s_DeviceState, ' LINK_WITHOUT_COMM B');
		66:
			visu_Data.st_Slave[i].s_DeviceState := CONCAT(visu_Data.st_Slave[i].s_DeviceState, ' LINK_WITHOUT_COMM C');
		130:
			visu_Data.st_Slave[i].s_DeviceState := CONCAT(visu_Data.st_Slave[i].s_DeviceState, ' LINK_WITHOUT_COMM D');
			
		20:
			visu_Data.st_Slave[i].s_DeviceState := CONCAT(visu_Data.st_Slave[i].s_DeviceState, ' MISSING_LINK A');
		36:
			visu_Data.st_Slave[i].s_DeviceState := CONCAT(visu_Data.st_Slave[i].s_DeviceState, ' MISSING_LINK B');
		68:
			visu_Data.st_Slave[i].s_DeviceState := CONCAT(visu_Data.st_Slave[i].s_DeviceState, ' MISSING_LINK C');
		132:
			visu_Data.st_Slave[i].s_DeviceState := CONCAT(visu_Data.st_Slave[i].s_DeviceState, ' MISSING_LINK D');
			
		24:
			visu_Data.st_Slave[i].s_DeviceState := CONCAT(visu_Data.st_Slave[i].s_DeviceState, ' ADDITIONAL_LINK A');
		40:
			visu_Data.st_Slave[i].s_DeviceState := CONCAT(visu_Data.st_Slave[i].s_DeviceState, ' ADDITIONAL_LINK B');
		72:
			visu_Data.st_Slave[i].s_DeviceState := CONCAT(visu_Data.st_Slave[i].s_DeviceState, ' ADDITIONAL_LINK C');
		136:
			visu_Data.st_Slave[i].s_DeviceState := CONCAT(visu_Data.st_Slave[i].s_DeviceState, ' ADDITIONAL_LINK D');
		
		ELSE
			visu_Data.st_Slave[i].s_DeviceState := CONCAT(visu_Data.st_Slave[i].s_DeviceState, ' undefined');
	END_CASE
END_FOR
END_ACTION

(* POU EPT Lib/Funktionen/Checks/CheckBounds, ST *)
FUNCTION CheckBounds : DINT
VAR_INPUT
	index, lower, upper 	: DINT;
END_VAR
VAR
END_VAR
IF index<lower THEN
	CheckBounds_ErrCnt := CheckBounds_ErrCnt + 1;
	CheckBounds := lower;
ELSIF index>upper THEN
	CheckBounds_ErrCnt := CheckBounds_ErrCnt + 1;
	CheckBounds := upper;
ELSE
	CheckBounds := index;
END_IF
END_FUNCTION

(* POU EPT Lib/Funktionen/Checks/CheckDivByte, ST *)
FUNCTION CheckDivByte : BYTE
VAR_INPUT
	divisor			 	: BYTE;
END_VAR
VAR
END_VAR
IF divisor = 0 THEN
	CheckByteZeroDiv_ErrCnt := CheckByteZeroDiv_ErrCnt + 1;
	CheckDivByte := 1;
ELSE
	CheckDivByte := divisor;
END_IF
END_FUNCTION

(* POU EPT Lib/Funktionen/Checks/CheckDivDWord, ST *)
FUNCTION CheckDivDWord : DWORD
VAR_INPUT
	divisor				: DWORD;
END_VAR
VAR
END_VAR
IF divisor = 0 THEN
	CheckDWordZeroDiv_ErrCnt := CheckDWordZeroDiv_ErrCnt + 1;
	CheckDivDWord := 1;
ELSE
	CheckDivDWord := divisor;
END_IF
END_FUNCTION

(* POU EPT Lib/Funktionen/Checks/CheckDivReal, ST *)
FUNCTION CheckDivReal : REAL
VAR_INPUT
	divisor		 		: REAL;
END_VAR
VAR
END_VAR
IF divisor = 0 THEN
	CheckRealZeroDiv_ErrCnt := CheckRealZeroDiv_ErrCnt + 1;
	CheckDivReal := 1;
ELSE
	CheckDivReal := divisor;
END_IF
END_FUNCTION

(* POU EPT Lib/Funktionen/Checks/CheckDivWord, ST *)
FUNCTION CheckDivWord : WORD
VAR_INPUT
	divisor				: WORD;
END_VAR
VAR
END_VAR
IF divisor = 0 THEN
	CheckWordZeroDiv_ErrCnt:= CheckWordZeroDiv_ErrCnt + 1;
	CheckDivWord := 1;
ELSE
	CheckDivWord := divisor;
END_IF
END_FUNCTION

(* POU EPT Lib/Funktionen/Checks/CheckRangeSigned, ST *)
FUNCTION CheckRangeSigned : DINT
VAR_INPUT
    value, lower, upper: DINT;
END_VAR
VAR
END_VAR
IF (value < lower) THEN
	CheckRangeSigned_ErrCnt := CheckRangeSigned_ErrCnt + 1;
	CheckRangeSigned := lower;
ELSIF(value > upper) THEN
	CheckRangeSigned_ErrCnt := CheckRangeSigned_ErrCnt + 1;
	CheckRangeSigned := upper;
ELSE
	CheckRangeSigned := value;
END_IF
END_FUNCTION

(* POU EPT Lib/Funktionen/Checks/CheckRangeUnsigned, ST *)
FUNCTION CheckRangeUnsigned : UDINT
VAR_INPUT
    value, lower, upper: UDINT;
END_VAR
VAR
END_VAR
IF (value < lower) THEN
	CheckRangeUnSigned_ErrCnt := CheckRangeUnsigned_ErrCnt + 1;
	CheckRangeUnsigned := lower;
ELSIF(value > upper) THEN
	CheckRangeUnsigned_ErrCnt := CheckRangeUnsigned_ErrCnt + 1;
	CheckRangeUnsigned := upper;
ELSE
	CheckRangeUnsigned := value;
END_IF
END_FUNCTION

(* POU EPT Lib/Funktionen/BOOLARRAY_TO_BYTE, ST *)
FUNCTION BOOLARRAY_TO_BYTE : BYTE
VAR_INPUT
	p_adr_buffer			: POINTER TO ARRAY[0..7] OF BOOL;
END_VAR
VAR
	tmp_buffer			: ARRAY[0..7] OF BOOL;
	tmp_byte				: BYTE;
	i16_index			: INT;
END_VAR
(* Aus einem Boolarray, soll ein Byte entstehen *)
tmp_buffer := p_adr_buffer^;

tmp_byte := 2#0;

FOR i16_index := 7 TO 0 BY -1 DO
	tmp_byte := tmp_byte OR BOOL_TO_BYTE(tmp_buffer[i16_index]);
	IF i16_index > 0 THEN
		tmp_byte := SHL(tmp_byte, 1);
	END_IF
END_FOR;

BOOLARRAY_TO_BYTE := tmp_byte; (* Rückgabewert der Funktion *)
END_FUNCTION

(* POU EPT Lib/Funktionen/BOOLARRAY_TO_DWORD, ST *)
FUNCTION BOOLARRAY_TO_DWORD : DWORD
VAR_INPUT
	p_adr_buffer			: POINTER TO ARRAY[0..31] OF BOOL;
END_VAR
VAR
	tmp_buffer			: ARRAY[0..31] OF BOOL;
	tmp_dword			: DWORD;
	i16_index			: INT;
END_VAR
(* Aus einem Boolarray, soll ein Doppelword entstehen *)
tmp_buffer := p_adr_buffer^;

tmp_dword := 2#0;

FOR i16_index := 31 TO 0 BY -1 DO
	tmp_dword := tmp_dword OR BOOL_TO_DWORD(tmp_buffer[i16_index]);
	IF i16_index > 0 THEN
		tmp_dword := SHL(tmp_dword, 1);
	END_IF
END_FOR;

BOOLARRAY_TO_DWORD := tmp_dword; (* Rückgabewert der Funktion *)
END_FUNCTION

(* POU EPT Lib/Funktionen/BOOLARRAY_TO_WORD, ST *)
FUNCTION BOOLARRAY_TO_WORD : WORD
VAR_INPUT
	p_adr_buffer			: POINTER TO ARRAY[0..15] OF BOOL;
END_VAR
VAR
	tmp_buffer			: ARRAY[0..15] OF BOOL;
	tmp_word			: WORD;
	i16_index			: INT;
END_VAR
(* Aus einem Boolarray, soll ein Word entstehen *)
tmp_buffer := p_adr_buffer^;

tmp_word := 2#0;

FOR i16_index := 15 TO 0 BY -1 DO
	tmp_word := tmp_word OR BOOL_TO_WORD(tmp_buffer[i16_index]);
	IF i16_index > 0 THEN
		tmp_word := SHL(tmp_word, 1);
	END_IF
END_FOR;

BOOLARRAY_TO_WORD := tmp_word; (* Rückgabewert der Funktion *)
END_FUNCTION

(* POU EPT Lib/Funktionen/BYTEARRAY_TO_STRING_WITH_DELIMITER, ST *)
FUNCTION BYTEARRAY_TO_STRING_WITH_DELIMITER : STRING
VAR_INPUT
	p_adr_buffer			: POINTER TO ARRAY[0..100] OF BYTE;
	i16_buffer_laenge		: INT;
	str_delimiter			: STRING; (* Punkt zum trennen der einzelnen Zahlen in der Net-Adresse *)
END_VAR
VAR
	tmp_buffer			: ARRAY[0..100] OF BYTE;
	tmp_string			: STRING;
	i16_index			: INT;
END_VAR
(* Aus einem Bytearray, welches die einzelnen Zahlen der Net-Adresse beinhaltet wird ein String erzeugt, welcher die Zahlen getrennt durch Punkte enthält *)
tmp_buffer := p_adr_buffer^;

tmp_string := ''; (* leerer String *)
FOR i16_index := 0 TO i16_buffer_laenge - 1 DO
	tmp_string :=CONCAT(tmp_string ,BYTE_TO_STRING(tmp_buffer[i16_index]));
	IF i16_index < i16_buffer_laenge - 1 THEN
		tmp_string := CONCAT(tmp_string,str_delimiter); (* "Punkt" einfügen in den String *)
	END_IF;
END_FOR;

BYTEARRAY_TO_STRING_WITH_DELIMITER := tmp_string; (* Rückgabewert der Funktion *)
END_FUNCTION

(* POU EPT Lib/Funktionen/F_Vergleich_Real, ST *)
FUNCTION F_Vergleich_Real : BOOL
VAR_INPUT
	r_wert			: REAL;
	r_vergleichswert	: REAL;
END_VAR
VAR
	r_toleranz		: REAL := 0.001;
END_VAR
IF ABS(r_wert - r_vergleichswert) < r_toleranz THEN
	F_Vergleich_Real := TRUE;
ELSE
	F_Vergleich_Real := FALSE;
END_IF
END_FUNCTION

(* POU EPT Lib/Funktionen/Scale, ST *)
FUNCTION Scale : REAL
VAR_INPUT
	i16Messwert : INT;
	i16MessbereichUnten : INT;
	i16MessbereichOben : INT;
	rSkaleUnten : REAL;
	rSkaleOben : REAL;
END_VAR
VAR
END_VAR
(* Überwachung auf Division durch Null*)
IF i16MessbereichOben <> i16MessbereichUnten THEN

Scale := ( rSkaleOben - rSkaleUnten ) * i16Messwert / ( i16MessbereichOben - i16MessbereichUnten );

END_IF
END_FUNCTION

(* POU EPT Lib/Funktionen/WORD_TO_BOOLARRAY, ST *)
FUNCTION WORD_TO_BOOLARRAY : ARRAY[0..15] OF BOOL
VAR_INPUT
	p_inputword			: WORD;
END_VAR
VAR
	tmp_bytearray		: ARRAY[0..15] OF BOOL;
	tmp_word			: WORD;
	i16_index			: INT;
END_VAR
(* Aus einem Word, soll ein Boolarray entstehen *)
tmp_word := p_inputword;

FOR i16_index := 15 TO 0 BY -1 DO
	tmp_bytearray[i16_index] := WORD_TO_BOOL(tmp_word AND 16#8000);
	tmp_word := SHL(tmp_word, 1);
END_FOR;

WORD_TO_BOOLARRAY := tmp_bytearray; (* Rückgabewert der Funktion *)
END_FUNCTION

(* POU EPT Lib/Funktionen/WORD_TO_STR_LEN, ST *)
FUNCTION WORD_TO_STR_LEN :STRING(255)
VAR_INPUT
	w_In		:WORD;
	i_Len		:INT:=1;
END_VAR

VAR
	i			:INT;
	i_LenIn		:INT;
	s_Help		:STRING(255);

END_VAR
(*
der INT Wert wird in einen String umgewandelt und mit 0 aufgefüllt oder 
abgeschnitten auf die deffinierte Länge *)

s_Help:=WORD_TO_STRING(w_In);
i_LenIn:=LEN(s_Help);

IF	i_LenIn < i_Len THEN
	FOR i := 1 TO i_Len - i_LenIn DO
		s_Help:=CONCAT('0',s_Help);
	END_FOR

ELSIF
	i_LenIn > i_Len THEN
	s_Help:=RIGHT(s_Help,i_Len);
END_IF

WORD_TO_STR_LEN:=s_Help;
END_FUNCTION

(* POU EPT Lib/Funktionsbausteine/Nockenschaltwerke/NSW_INT/ST_Nockenschaltwerk_int, ST *)
FUNCTION_BLOCK ST_Nockenschaltwerk_int
VAR_INPUT
	i16_achsposition							: INT;
	i16_achsgeschwindigkeit					: INT;
	st_config									: struct_config;
END_VAR
VAR_IN_OUT
	st_visu									: struct_visu;
	arr_nocken								: ARRAY [0..15] OF struct_nocken_int;
END_VAR
VAR_OUTPUT
END_VAR
VAR
	b_first_cycle 								: BOOL := TRUE;
	i16_aktuelle_pos 							: INT := 0;
	i16_alte_pos	 							: INT := 0;
	r_zeit_fuer_1einheit						: REAL := 0.0;
	i16_anfangspos_mit_tzk 					: ARRAY [0..15] OF INT := 0;
	i16_endpos_mit_tzk 						: ARRAY [0..15] OF INT := 0;
	i16_vorsteuerpos_max						: INT := 0;
	b_verfahrrichtung_positiv 					: BOOL := FALSE;
	b_verfahrrichtung_negativ					: BOOL := FALSE;
	sm_positionseingabe						: BOOL := FALSE;
	sm_vorsteuerung							: BOOL := FALSE;
	sp, no									: UINT := 0;
	arr_spur									: ARRAY [0..15] OF BOOL;
	b_setzustand_anfang_kleiner_ende			: ARRAY [0..15] OF BOOL;
	b_setzustand_anfang_groesser_ende		: ARRAY [0..15] OF BOOL;
	b_resetzustand_anfang_kleiner_ende		: ARRAY [0..15] OF BOOL;
	b_resetzustand_anfang_groesser_ende		: ARRAY [0..15] OF BOOL;
END_VAR
(* Funktionsbaustein Nockenschaltwerk *)
IF b_first_cycle THEN
	b_first_cycle := FALSE;
	i16_vorsteuerpos_max := 60;
	b_verfahrrichtung_positiv := TRUE;
	b_verfahrrichtung_negativ := FALSE;
	i16_alte_pos := i16_aktuelle_pos;
END_IF

(* Aktuelle Position für weitere Komponenten zur Verfügung stellen *)
i16_aktuelle_pos := i16_achsposition;

(* Verfahrrichtung überwachen *)
IF i16_aktuelle_pos > i16_alte_pos THEN
	b_verfahrrichtung_positiv := TRUE;
	b_verfahrrichtung_negativ := FALSE;
	i16_alte_pos := i16_aktuelle_pos;
ELSIF i16_aktuelle_pos < i16_alte_pos THEN
	b_verfahrrichtung_positiv := FALSE;
	b_verfahrrichtung_negativ := TRUE;
	i16_alte_pos := i16_aktuelle_pos;
END_IF

IF i16_achsgeschwindigkeit >= 1 THEN
	(* 0.006 = 360Grad / (60sec * 1000ms) *)
	r_zeit_fuer_1einheit := 0.006 * INT_TO_REAL(i16_achsgeschwindigkeit);	(* REAL-Zahl in ms *)
ELSE
	r_zeit_fuer_1einheit := 0.0;
END_IF

(* Erst alle Spuren reset *)
FOR sp := 0  TO SIZEOF (arr_spur)/SIZEOF(arr_spur[0]) - 1BY 1 DO
	arr_spur[sp] :=FALSE;
END_FOR

(* Totzeitkompensation durch Vorsteuerung *)
FOR no := 0  TO SIZEOF (arr_nocken)/SIZEOF(arr_nocken[0]) - 1 BY 1DO
	(* Berechnung des Vorsteuerwinkels *)
	arr_nocken[no].i16_vorsteuerpos :=  REAL_TO_INT((TIME_TO_REAL(arr_nocken[no].t_vorsteuerzeit)) * r_zeit_fuer_1einheit);
	IF  arr_nocken[no].i16_vorsteuerpos >=i16_vorsteuerpos_max THEN
		 arr_nocken[no].i16_vorsteuerpos := 0;
		sm_vorsteuerung := TRUE;
	ELSE
		sm_vorsteuerung := FALSE;
	END_IF

	(* Nockentoleranz mit Berücksichtigung der Vorsteuerzeit für Anfangswinkel*)
	i16_anfangspos_mit_tzk[no] := arr_nocken[no].i16_cam_begin -  arr_nocken[no].i16_vorsteuerpos;
	IF i16_anfangspos_mit_tzk[no] > 360 THEN
		i16_anfangspos_mit_tzk[no] := i16_anfangspos_mit_tzk[no] - 360;
	ELSIF i16_anfangspos_mit_tzk[no] < 0 THEN
		i16_anfangspos_mit_tzk[no] := i16_anfangspos_mit_tzk[no] + 360;
	END_IF
	(* Nockentoleranz mit Berücksichtigung der Vorsteuerzeit für Endwinkel*)
	i16_endpos_mit_tzk[no] := arr_nocken[no].i16_cam_end -  arr_nocken[no].i16_vorsteuerpos;
	IF i16_endpos_mit_tzk[no] > 360 THEN
		i16_endpos_mit_tzk[no] := i16_endpos_mit_tzk[no] - 360;
	ELSIF i16_endpos_mit_tzk[no] < 0 THEN
		i16_endpos_mit_tzk[no] := i16_endpos_mit_tzk[no] + 360;
	END_IF

